// TIA Portal V20 program export: 3 tag tables, 2 data types, 1 data blocks, 4 code blocks (in call order from the OBs), 4 instance data blocks

VAR_GLOBAL   // PLC tag table "IO_Device_PCL_Centralilze_PLC_Functinal_Test_1"
   In_Test_Parameters AT %I100.0 : "IO_Device_Test_Parameters";
   Out_Functinal_Test AT %Q100.0 : "IO_Device_Functinal_Test";
   Voltage_Read_UInt AT %QW160 : UInt;
END_VAR

VAR_GLOBAL   // PLC tag table "IO_PLC_Functinal_Test_1_PLC_Functinal_Test_3"
   In_Functional_Test AT %I300.0 : "IO_Device_Functinal_Test";
   Out_Test_Parameters AT %Q300.0 : "IO_Device_Test_Parameters";
END_VAR

VAR_GLOBAL   // PLC tag table "PLC_Functional_Test"
   Button_Start_Approve AT %I0.0 : Bool;
   Digital_Input_1 AT %I0.1 : Bool;
   Digital_Input_2 AT %I0.2 : Bool;
   Digital_Input_3 AT %I0.3 : Bool;
   Digital_Input_4 AT %I0.4 : Bool;
   Digital_Input_5 AT %I0.5 : Bool;
   Current_Transducer AT %IW64 : Int;
   Voltage_Transducer AT %IW66 : Int;
   Button_Light AT %Q0.0 : Bool;
   Light_Fail_Test AT %Q0.1 : Bool;
   Light_Approve_Test AT %Q0.2 : Bool;
   Digital_Output_3 AT %Q0.3 : Bool;
   Clock_Byte AT %MB0 : Byte;
   Clock_10Hz AT %M0.0 : Bool;
   Clock_5Hz AT %M0.1 : Bool;
   "Clock_2.5Hz" AT %M0.2 : Bool;
   Clock_2Hz AT %M0.3 : Bool;
   "Clock_1.25Hz" AT %M0.4 : Bool;
   Clock_1Hz AT %M0.5 : Bool;
   "Clock_0.625Hz" AT %M0.6 : Bool;
   "Clock_0.5Hz" AT %M0.7 : Bool;
   System_Byte AT %MB1 : Byte;
   FirstScan AT %M1.0 : Bool;
   DiagStatusUpdate AT %M1.1 : Bool;
   AlwaysTRUE AT %M1.2 : Bool;
   AlwaysFALSE AT %M1.3 : Bool;
END_VAR

TYPE "IO_Device_Functinal_Test"
   STRUCT
      Life_Trigger_PLC_Functional_Test_1 : Bool;
      Star_Test_PLC_Functional_Test_1 : Bool;
      Button_PLC_Functional_Test_1 : Bool;
      Electrical_Current_Test_Approved_PLC_Functional_Test_1 : Bool;
      Visual_Test_Approved_PLC_Functional_Test_1 : Bool;
      Electrical_Current_Read_PLC_Functional_Test_1 : UInt;
      Life_Trigger_PLC_Functional_Test_3 : Bool;
      Star_Test_PLC_Functional_Test_3 : Bool;
      Button_PLC_Functional_Test_3 : Bool;
      Electrical_Current_Test_Approved_PLC_Functional_Test_3 : Bool;
      Visual_Test_Approved_PLC_Functional_Test_3 : Bool;
      Electrical_Current_Read_PLC_Functional_Test_3 : UInt;
      Life_Trigger_PLC_Functional_Test_5 : Bool;
      Star_Test_PLC_Functional_Test_5 : Bool;
      Button_PLC_Functional_Test_5 : Bool;
      Electrical_Current_Test_Approved_PLC_Functional_Test_5 : Bool;
      Visual_Test_Approved_PLC_Functional_Test_5 : Bool;
      Electrical_Current_Read_PLC_Functional_Test_5 : UInt;
      Life_Trigger_PLC_Functional_Test_7 : Bool;
      Star_Test_PLC_Functional_Test_7 : Bool;
      Button_PLC_Functional_Test_7 : Bool;
      Electrical_Current_Test_Approved_PLC_Functional_Test_7 : Bool;
      Visual_Test_Approved_PLC_Functional_Test_7 : Bool;
      Electrical_Current_Read_PLC_Functional_Test_7 : UInt;
      Life_Trigger_PLC_Functional_Test_9 : Bool;
      Star_Test_PLC_Functional_Test_9 : Bool;
      Button_PLC_Functional_Test_9 : Bool;
      Electrical_Current_Test_Approved_PLC_Functional_Test_9 : Bool;
      Visual_Test_Approved_PLC_Functional_Test_9 : Bool;
      Electrical_Current_Read_PLC_Functional_Test_9 : UInt;
      Life_Trigger_PLC_Functional_Test_11 : Bool;
      Star_Test_PLC_Functional_Test_11 : Bool;
      Button_PLC_Functional_Test_11 : Bool;
      Electrical_Current_Test_Approved_PLC_Functional_Test_11 : Bool;
      Visual_Test_Approved_PLC_Functional_Test_11 : Bool;
      Electrical_Current_Read_PLC_Functional_Test_11 : UInt;
      Life_Trigger_PLC_Functional_Test_13 : Bool;
      Star_Test_PLC_Functional_Test_13 : Bool;
      Button_PLC_Functional_Test_13 : Bool;
      Electrical_Current_Test_Approved_PLC_Functional_Test_13 : Bool;
      Visual_Test_Approved_PLC_Functional_Test_13 : Bool;
      Electrical_Current_Read_PLC_Functional_Test_13 : UInt;
      Life_Trigger_PLC_Functional_Test_15 : Bool;
      Star_Test_PLC_Functional_Test_15 : Bool;
      Button_PLC_Functional_Test_15 : Bool;
      Electrical_Current_Test_Approved_PLC_Functional_Test_15 : Bool;
      Visual_Test_Approved_PLC_Functional_Test_15 : Bool;
      Electrical_Current_Read_PLC_Functional_Test_15 : UInt;
      Life_Trigger_PLC_Functional_Test_17 : Bool;
      Star_Test_PLC_Functional_Test_17 : Bool;
      Button_PLC_Functional_Test_17 : Bool;
      Electrical_Current_Test_Approved_PLC_Functional_Test_17 : Bool;
      Visual_Test_Approved_PLC_Functional_Test_17 : Bool;
      Electrical_Current_Read_PLC_Functional_Test_17 : UInt;
      Life_Trigger_PLC_Functional_Test_19 : Bool;
      Star_Test_PLC_Functional_Test_19 : Bool;
      Button_PLC_Functional_Test_19 : Bool;
      Electrical_Current_Test_Approved_PLC_Functional_Test_19 : Bool;
      Visual_Test_Approved_PLC_Functional_Test_19 : Bool;
      Electrical_Current_Read_PLC_Functional_Test_19 : UInt;
      Life_Trigger_PLC_Functional_Test_21 : Bool;
      Star_Test_PLC_Functional_Test_21 : Bool;
      Button_PLC_Functional_Test_21 : Bool;
      Electrical_Current_Test_Approved_PLC_Functional_Test_21 : Bool;
      Visual_Test_Approved_PLC_Functional_Test_21 : Bool;
      Electrical_Current_Read_PLC_Functional_Test_21 : UInt;
      Life_Trigger_PLC_Functional_Test_23 : Bool;
      Star_Test_PLC_Functional_Test_23 : Bool;
      Button_PLC_Functional_Test_23 : Bool;
      Electrical_Current_Test_Approved_PLC_Functional_Test_23 : Bool;
      Visual_Test_Approved_PLC_Functional_Test_23 : Bool;
      Electrical_Current_Read_PLC_Functional_Test_23 : UInt;
      Life_Trigger_PLC_Functional_Test_25 : Bool;
      Star_Test_PLC_Functional_Test_25 : Bool;
      Button_PLC_Functional_Test_25 : Bool;
      Electrical_Current_Test_Approved_PLC_Functional_Test_25 : Bool;
      Visual_Test_Approved_PLC_Functional_Test_25 : Bool;
      Electrical_Current_Read_PLC_Functional_Test_25 : UInt;
      Life_Trigger_PLC_Functional_Test_27 : Bool;
      Star_Test_PLC_Functional_Test_27 : Bool;
      Button_PLC_Functional_Test_27 : Bool;
      Electrical_Current_Test_Approved_PLC_Functional_Test_27 : Bool;
      Visual_Test_Approved_PLC_Functional_Test_27 : Bool;
      Electrical_Current_Read_PLC_Functional_Test_27 : UInt;
      Life_Trigger_PLC_Functional_Test_29 : Bool;
      Star_Test_PLC_Functional_Test_29 : Bool;
      Button_PLC_Functional_Test_29 : Bool;
      Electrical_Current_Test_Approved_PLC_Functional_Test_29 : Bool;
      Visual_Test_Approved_PLC_Functional_Test_29 : Bool;
      Electrical_Current_Read_PLC_Functional_Test_29 : UInt;
   END_STRUCT;
END_TYPE

TYPE "IO_Device_Test_Parameters"
   STRUCT
      Reset_PLC_Functional_Test_1 : Bool;
      Reset_PLC_Functional_Test_3 : Bool;
      Reset_PLC_Functional_Test_5 : Bool;
      Reset_PLC_Functional_Test_7 : Bool;
      Reset_PLC_Functional_Test_9 : Bool;
      Reset_PLC_Functional_Test_11 : Bool;
      Reset_PLC_Functional_Test_13 : Bool;
      Reset_PLC_Functional_Test_15 : Bool;
      Reset_PLC_Functional_Test_17 : Bool;
      Reset_PLC_Functional_Test_19 : Bool;
      Reset_PLC_Functional_Test_21 : Bool;
      Reset_PLC_Functional_Test_23 : Bool;
      Reset_PLC_Functional_Test_25 : Bool;
      Reset_PLC_Functional_Test_27 : Bool;
      Reset_PLC_Functional_Test_29 : Bool;
      Status : Bool;
      Voltage_Read : UInt;
      Min_Electrical_Current : UInt;
      Max_Electrical_Current : UInt;
      Time_End_Electrical_Current_Test : Time;
      Time_Start_Visual_Test : Time;
   END_STRUCT;
END_TYPE

DATA_BLOCK "DB_Test_Water_Foutain"   // DB4
{ S7_Optimized_Access := 'TRUE' }
// stored: MemoryReserve 100
   VAR
      Star_Functional_Test : Bool;
      Reset_Functional_Test : Bool;
      Electrical_Current_Test_Approved : Bool;
      Visual_Test_Approved_PLC : Bool;
   END_VAR
BEGIN
END_DATA_BLOCK

ORGANIZATION_BLOCK "Main"   // OB1, LAD, ProgramCycle
TITLE = "Main Program Sweep (Cycle)"
{ S7_Optimized_Access := 'TRUE' }
// stored: SetENOAutomatically false
   VAR_INPUT
      Initial_Call : Bool;   // Initial call of this OB
      Remanence : Bool;   // =True, if remanent data are available
   END_VAR
   VAR CONSTANT
      Test_Station : SInt := 1;
      Total_Number_Test_Stations : SInt := 25;
   END_VAR
BEGIN

REGION Network 1: Digital Inputs
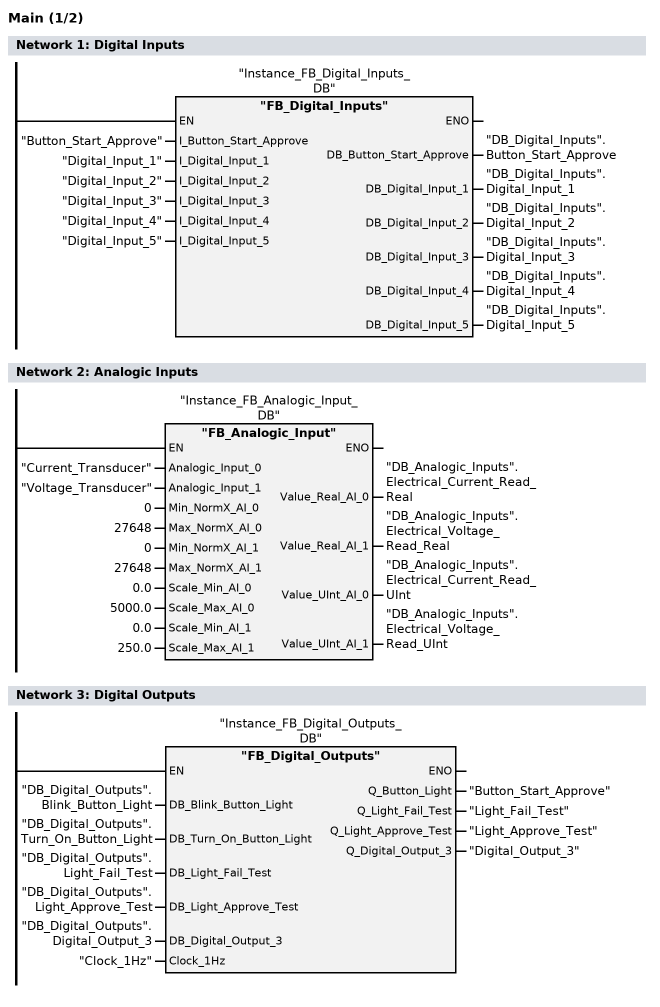
   RUNG wire#powerrail
      "Instance_FB_Digital_Inputs_DB"(I_Button_Start_Approve := "Button_Start_Approve", I_Digital_Input_1 := "Digital_Input_1", I_Digital_Input_2 := "Digital_Input_2", I_Digital_Input_3 := "Digital_Input_3", I_Digital_Input_4 := "Digital_Input_4", I_Digital_Input_5 := "Digital_Input_5", DB_Button_Start_Approve => "DB_Digital_Inputs".Button_Start_Approve, DB_Digital_Input_1 => "DB_Digital_Inputs".Digital_Input_1, DB_Digital_Input_2 => "DB_Digital_Inputs".Digital_Input_2, DB_Digital_Input_3 => "DB_Digital_Inputs".Digital_Input_3, DB_Digital_Input_4 => "DB_Digital_Inputs".Digital_Input_4, DB_Digital_Input_5 => "DB_Digital_Inputs".Digital_Input_5)
   END_RUNG
   // the same network as SCL:
   "Instance_FB_Digital_Inputs_DB"(I_Button_Start_Approve := "Button_Start_Approve",   // "FB_Digital_Inputs"
                           I_Digital_Input_1 := "Digital_Input_1",
                           I_Digital_Input_2 := "Digital_Input_2",
                           I_Digital_Input_3 := "Digital_Input_3",
                           I_Digital_Input_4 := "Digital_Input_4",
                           I_Digital_Input_5 := "Digital_Input_5",
                           DB_Button_Start_Approve => "DB_Digital_Inputs".Button_Start_Approve,
                           DB_Digital_Input_1 => "DB_Digital_Inputs".Digital_Input_1,
                           DB_Digital_Input_2 => "DB_Digital_Inputs".Digital_Input_2,
                           DB_Digital_Input_3 => "DB_Digital_Inputs".Digital_Input_3,
                           DB_Digital_Input_4 => "DB_Digital_Inputs".Digital_Input_4,
                           DB_Digital_Input_5 => "DB_Digital_Inputs".Digital_Input_5);
END_REGION

REGION Network 2: Analogic Inputs
   RUNG wire#powerrail
      "Instance_FB_Analogic_Input_DB"(Analogic_Input_0 := "Current_Transducer", Analogic_Input_1 := "Voltage_Transducer", Min_NormX_AI_0 := 0, Max_NormX_AI_0 := 27648, Min_NormX_AI_1 := 0, Max_NormX_AI_1 := 27648, Scale_Min_AI_0 := 0.0, Scale_Max_AI_0 := 5000.0, Scale_Min_AI_1 := 0.0, Scale_Max_AI_1 := 250.0, Value_Real_AI_0 => "DB_Analogic_Inputs".Electrical_Current_Read_Real, Value_Real_AI_1 => "DB_Analogic_Inputs".Electrical_Voltage_Read_Real, Value_UInt_AI_0 => "DB_Analogic_Inputs".Electrical_Current_Read_UInt, Value_UInt_AI_1 => "DB_Analogic_Inputs".Electrical_Voltage_Read_UInt)
   END_RUNG
   // the same network as SCL:
   "Instance_FB_Analogic_Input_DB"(Analogic_Input_0 := "Current_Transducer",   // "FB_Analogic_Input"
                           Analogic_Input_1 := "Voltage_Transducer",
                           Min_NormX_AI_0 := 0,
                           Max_NormX_AI_0 := 27648,
                           Min_NormX_AI_1 := 0,
                           Max_NormX_AI_1 := 27648,
                           Scale_Min_AI_0 := 0.0,
                           Scale_Max_AI_0 := 5000.0,
                           Scale_Min_AI_1 := 0.0,
                           Scale_Max_AI_1 := 250.0,
                           Value_Real_AI_0 => "DB_Analogic_Inputs".Electrical_Current_Read_Real,
                           Value_Real_AI_1 => "DB_Analogic_Inputs".Electrical_Voltage_Read_Real,
                           Value_UInt_AI_0 => "DB_Analogic_Inputs".Electrical_Current_Read_UInt,
                           Value_UInt_AI_1 => "DB_Analogic_Inputs".Electrical_Voltage_Read_UInt);
END_REGION

REGION Network 3: Digital Outputs
   RUNG wire#powerrail
      "Instance_FB_Digital_Outputs_DB"(DB_Blink_Button_Light := "DB_Digital_Outputs".Blink_Button_Light, DB_Turn_On_Button_Light := "DB_Digital_Outputs".Turn_On_Button_Light, DB_Light_Fail_Test := "DB_Digital_Outputs".Light_Fail_Test, DB_Light_Approve_Test := "DB_Digital_Outputs".Light_Approve_Test, DB_Digital_Output_3 := "DB_Digital_Outputs".Digital_Output_3, Clock_1Hz := "Clock_1Hz", Q_Button_Light => "Button_Start_Approve", Q_Light_Fail_Test => "Light_Fail_Test", Q_Light_Approve_Test => "Light_Approve_Test", Q_Digital_Output_3 => "Digital_Output_3")
   END_RUNG
   // the same network as SCL:
   "Instance_FB_Digital_Outputs_DB"(DB_Blink_Button_Light := "DB_Digital_Outputs".Blink_Button_Light,   // "FB_Digital_Outputs"
                           DB_Turn_On_Button_Light := "DB_Digital_Outputs".Turn_On_Button_Light,
                           DB_Light_Fail_Test := "DB_Digital_Outputs".Light_Fail_Test,
                           DB_Light_Approve_Test := "DB_Digital_Outputs".Light_Approve_Test,
                           DB_Digital_Output_3 := "DB_Digital_Outputs".Digital_Output_3,
                           Clock_1Hz := "Clock_1Hz",
                           Q_Button_Light => "Button_Start_Approve",
                           Q_Light_Fail_Test => "Light_Fail_Test",
                           Q_Light_Approve_Test => "Light_Approve_Test",
                           Q_Digital_Output_3 => "Digital_Output_3");
END_REGION

REGION Network 4: IO Device
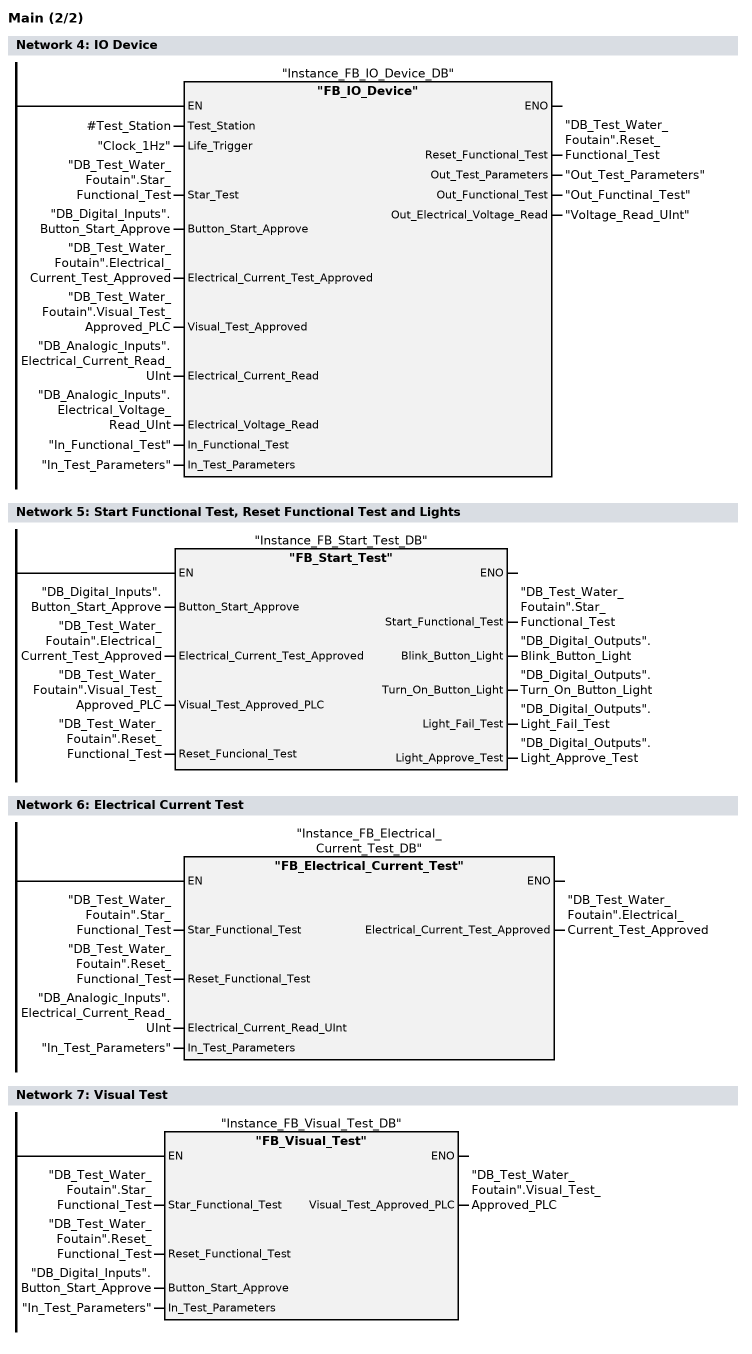
   RUNG wire#powerrail
      "Instance_FB_IO_Device_DB"(Test_Station := #Test_Station, Life_Trigger := "Clock_1Hz", Star_Test := "DB_Test_Water_Foutain".Star_Functional_Test, Button_Start_Approve := "DB_Digital_Inputs".Button_Start_Approve, Electrical_Current_Test_Approved := "DB_Test_Water_Foutain".Electrical_Current_Test_Approved, Visual_Test_Approved := "DB_Test_Water_Foutain".Visual_Test_Approved_PLC, Electrical_Current_Read := "DB_Analogic_Inputs".Electrical_Current_Read_UInt, Electrical_Voltage_Read := "DB_Analogic_Inputs".Electrical_Voltage_Read_UInt, In_Functional_Test := "In_Functional_Test", In_Test_Parameters := "In_Test_Parameters", Reset_Functional_Test => "DB_Test_Water_Foutain".Reset_Functional_Test, Out_Test_Parameters => "Out_Test_Parameters", Out_Functional_Test => "Out_Functinal_Test", Out_Electrical_Voltage_Read => "Voltage_Read_UInt")
   END_RUNG
   // the same network as SCL:
   "Instance_FB_IO_Device_DB"(Test_Station := #Test_Station,   // "FB_IO_Device"
                           Life_Trigger := "Clock_1Hz",
                           Star_Test := "DB_Test_Water_Foutain".Star_Functional_Test,
                           Button_Start_Approve := "DB_Digital_Inputs".Button_Start_Approve,
                           Electrical_Current_Test_Approved := "DB_Test_Water_Foutain".Electrical_Current_Test_Approved,
                           Visual_Test_Approved := "DB_Test_Water_Foutain".Visual_Test_Approved_PLC,
                           Electrical_Current_Read := "DB_Analogic_Inputs".Electrical_Current_Read_UInt,
                           Electrical_Voltage_Read := "DB_Analogic_Inputs".Electrical_Voltage_Read_UInt,
                           In_Functional_Test := "In_Functional_Test",
                           In_Test_Parameters := "In_Test_Parameters",
                           Reset_Functional_Test => "DB_Test_Water_Foutain".Reset_Functional_Test,
                           Out_Test_Parameters => "Out_Test_Parameters",
                           Out_Functional_Test => "Out_Functinal_Test",
                           Out_Electrical_Voltage_Read => "Voltage_Read_UInt");
END_REGION

REGION Network 5: Start Functional Test, Reset Functional Test and Lights
   RUNG wire#powerrail
      "Instance_FB_Start_Test_DB"(Button_Start_Approve := "DB_Digital_Inputs".Button_Start_Approve, Electrical_Current_Test_Approved := "DB_Test_Water_Foutain".Electrical_Current_Test_Approved, Visual_Test_Approved_PLC := "DB_Test_Water_Foutain".Visual_Test_Approved_PLC, Reset_Funcional_Test := "DB_Test_Water_Foutain".Reset_Functional_Test, Start_Functional_Test => "DB_Test_Water_Foutain".Star_Functional_Test, Blink_Button_Light => "DB_Digital_Outputs".Blink_Button_Light, Turn_On_Button_Light => "DB_Digital_Outputs".Turn_On_Button_Light, Light_Fail_Test => "DB_Digital_Outputs".Light_Fail_Test, Light_Approve_Test => "DB_Digital_Outputs".Light_Approve_Test)
   END_RUNG
   // the same network as SCL:
   "Instance_FB_Start_Test_DB"(Button_Start_Approve := "DB_Digital_Inputs".Button_Start_Approve,   // "FB_Start_Test"
                           Electrical_Current_Test_Approved := "DB_Test_Water_Foutain".Electrical_Current_Test_Approved,
                           Visual_Test_Approved_PLC := "DB_Test_Water_Foutain".Visual_Test_Approved_PLC,
                           Reset_Funcional_Test := "DB_Test_Water_Foutain".Reset_Functional_Test,
                           Start_Functional_Test => "DB_Test_Water_Foutain".Star_Functional_Test,
                           Blink_Button_Light => "DB_Digital_Outputs".Blink_Button_Light,
                           Turn_On_Button_Light => "DB_Digital_Outputs".Turn_On_Button_Light,
                           Light_Fail_Test => "DB_Digital_Outputs".Light_Fail_Test,
                           Light_Approve_Test => "DB_Digital_Outputs".Light_Approve_Test);
END_REGION

REGION Network 6: Electrical Current Test
   RUNG wire#powerrail
      "Instance_FB_Electrical_Current_Test_DB"(Star_Functional_Test := "DB_Test_Water_Foutain".Star_Functional_Test, Reset_Functional_Test := "DB_Test_Water_Foutain".Reset_Functional_Test, Electrical_Current_Read_UInt := "DB_Analogic_Inputs".Electrical_Current_Read_UInt, In_Test_Parameters := "In_Test_Parameters", Electrical_Current_Test_Approved => "DB_Test_Water_Foutain".Electrical_Current_Test_Approved)
   END_RUNG
   // the same network as SCL:
   "Instance_FB_Electrical_Current_Test_DB"(Star_Functional_Test := "DB_Test_Water_Foutain".Star_Functional_Test,   // "FB_Electrical_Current_Test"
                           Reset_Functional_Test := "DB_Test_Water_Foutain".Reset_Functional_Test,
                           Electrical_Current_Read_UInt := "DB_Analogic_Inputs".Electrical_Current_Read_UInt,
                           In_Test_Parameters := "In_Test_Parameters",
                           Electrical_Current_Test_Approved => "DB_Test_Water_Foutain".Electrical_Current_Test_Approved);
END_REGION

REGION Network 7: Visual Test
   RUNG wire#powerrail
      "Instance_FB_Visual_Test_DB"(Star_Functional_Test := "DB_Test_Water_Foutain".Star_Functional_Test, Reset_Functional_Test := "DB_Test_Water_Foutain".Reset_Functional_Test, Button_Start_Approve := "DB_Digital_Inputs".Button_Start_Approve, In_Test_Parameters := "In_Test_Parameters", Visual_Test_Approved_PLC => "DB_Test_Water_Foutain".Visual_Test_Approved_PLC)
   END_RUNG
   // the same network as SCL:
   "Instance_FB_Visual_Test_DB"(Star_Functional_Test := "DB_Test_Water_Foutain".Star_Functional_Test,   // "FB_Visual_Test"
                           Reset_Functional_Test := "DB_Test_Water_Foutain".Reset_Functional_Test,
                           Button_Start_Approve := "DB_Digital_Inputs".Button_Start_Approve,
                           In_Test_Parameters := "In_Test_Parameters",
                           Visual_Test_Approved_PLC => "DB_Test_Water_Foutain".Visual_Test_Approved_PLC);
END_REGION
END_ORGANIZATION_BLOCK

FUNCTION_BLOCK "FB_IO_Device"   // FB4, LAD
{ S7_Optimized_Access := 'TRUE' }
// stored: MemoryReserve 100, SetENOAutomatically false
   VAR_INPUT
      Test_Station : SInt;
      Life_Trigger : Bool;
      Star_Test : Bool;
      Button_Start_Approve : Bool;
      Electrical_Current_Test_Approved : Bool;
      Visual_Test_Approved : Bool;
      Electrical_Current_Read : UInt;
      Electrical_Voltage_Read : UInt;
      In_Functional_Test : "IO_Device_Functinal_Test";
      In_Test_Parameters : "IO_Device_Test_Parameters";
   END_VAR
   VAR_OUTPUT
      Reset_Functional_Test : Bool;
      Out_Test_Parameters : "IO_Device_Test_Parameters";
      Out_Functional_Test : "IO_Device_Functinal_Test";
      Out_Electrical_Voltage_Read : UInt;
   END_VAR
   VAR_TEMP   // added for the SCL form of the ladder/FBD networks
      _w1 : Bool;
   END_VAR
BEGIN

REGION Network 1: Test Parameters
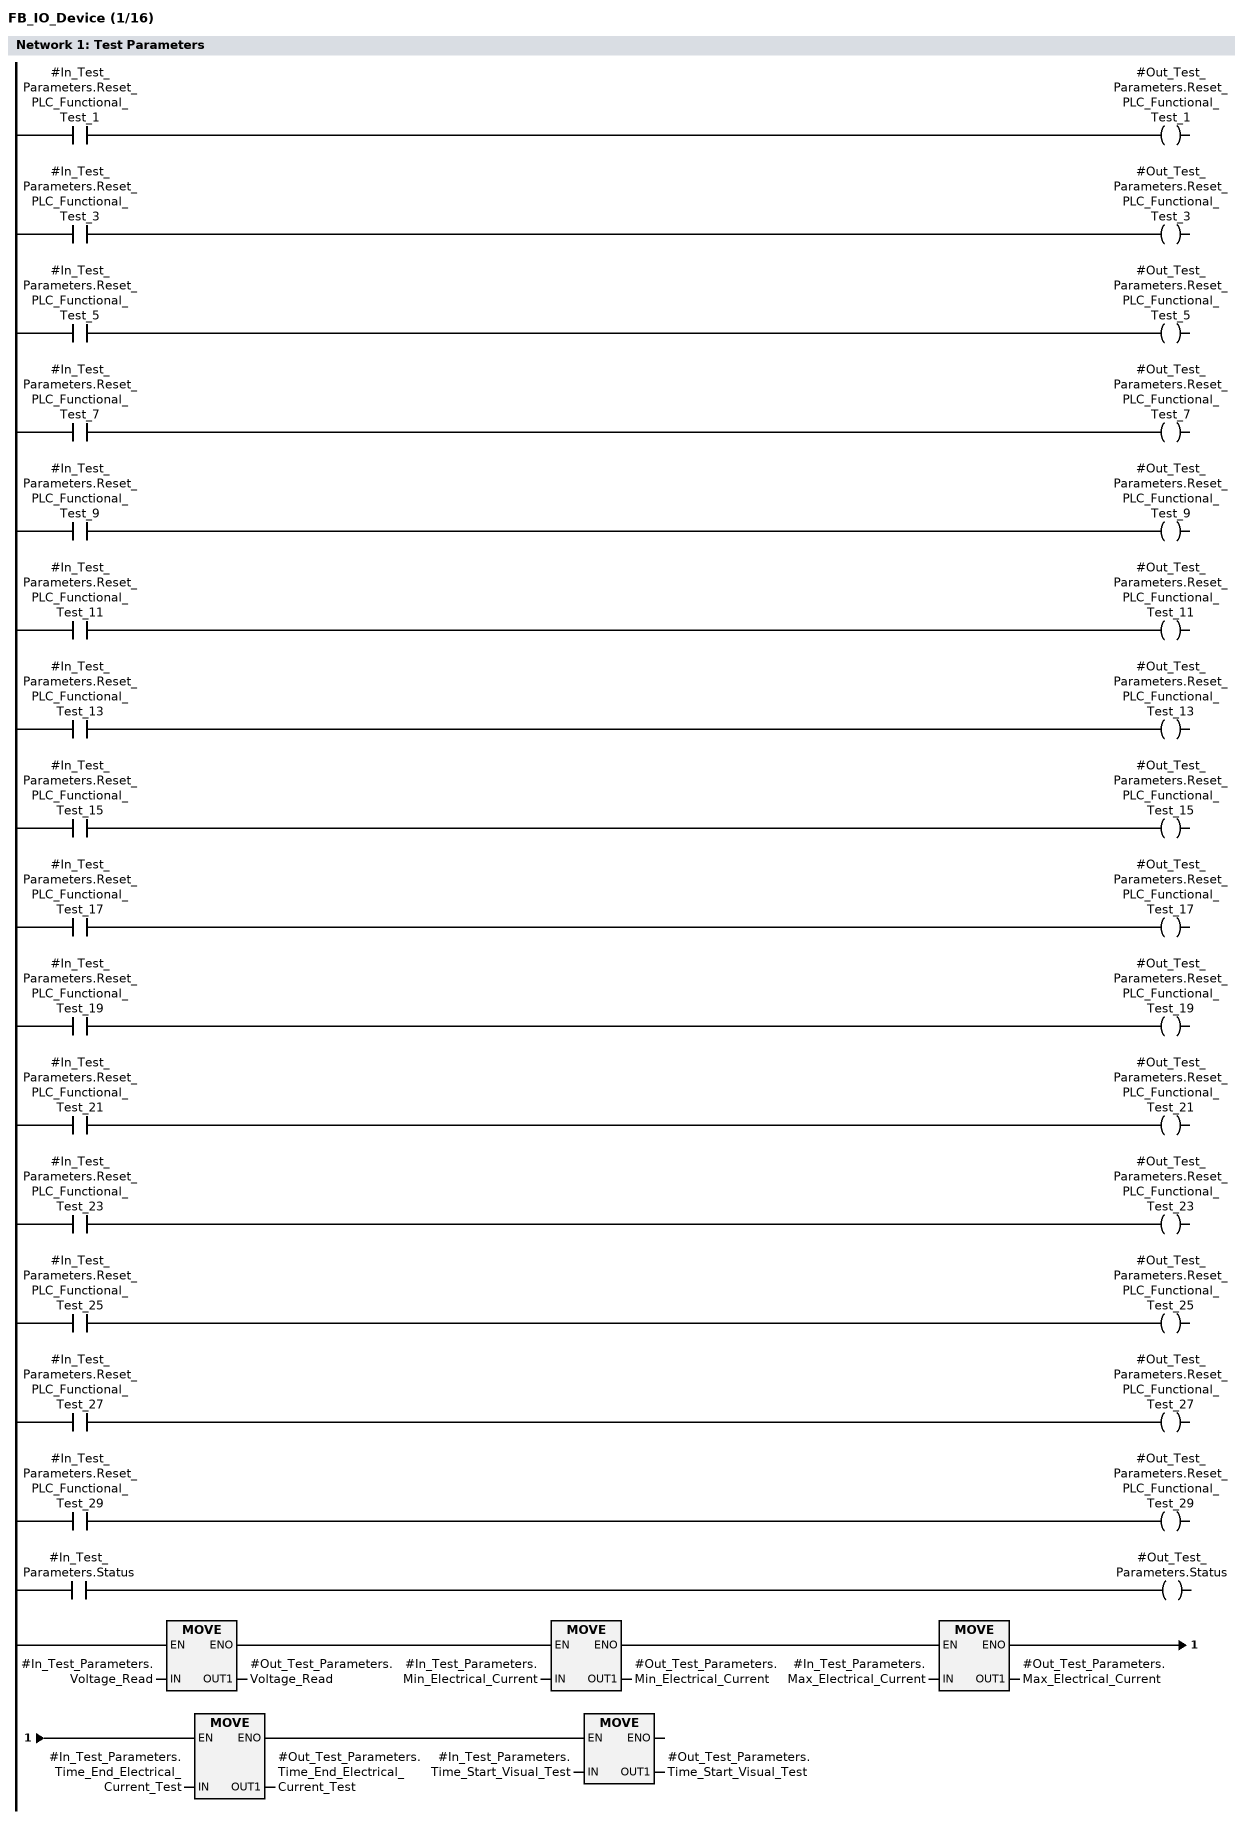
   RUNG wire#powerrail
      Contact( #In_Test_Parameters.Reset_PLC_Functional_Test_1 )
      Coil( #Out_Test_Parameters.Reset_PLC_Functional_Test_1 )
   END_RUNG
   RUNG wire#powerrail
      Contact( #In_Test_Parameters.Reset_PLC_Functional_Test_3 )
      Coil( #Out_Test_Parameters.Reset_PLC_Functional_Test_3 )
   END_RUNG
   RUNG wire#powerrail
      Contact( #In_Test_Parameters.Reset_PLC_Functional_Test_5 )
      Coil( #Out_Test_Parameters.Reset_PLC_Functional_Test_5 )
   END_RUNG
   RUNG wire#powerrail
      Contact( #In_Test_Parameters.Reset_PLC_Functional_Test_7 )
      Coil( #Out_Test_Parameters.Reset_PLC_Functional_Test_7 )
   END_RUNG
   RUNG wire#powerrail
      Contact( #In_Test_Parameters.Reset_PLC_Functional_Test_9 )
      Coil( #Out_Test_Parameters.Reset_PLC_Functional_Test_9 )
   END_RUNG
   RUNG wire#powerrail
      Contact( #In_Test_Parameters.Reset_PLC_Functional_Test_11 )
      Coil( #Out_Test_Parameters.Reset_PLC_Functional_Test_11 )
   END_RUNG
   RUNG wire#powerrail
      Contact( #In_Test_Parameters.Reset_PLC_Functional_Test_13 )
      Coil( #Out_Test_Parameters.Reset_PLC_Functional_Test_13 )
   END_RUNG
   RUNG wire#powerrail
      Contact( #In_Test_Parameters.Reset_PLC_Functional_Test_15 )
      Coil( #Out_Test_Parameters.Reset_PLC_Functional_Test_15 )
   END_RUNG
   RUNG wire#powerrail
      Contact( #In_Test_Parameters.Reset_PLC_Functional_Test_17 )
      Coil( #Out_Test_Parameters.Reset_PLC_Functional_Test_17 )
   END_RUNG
   RUNG wire#powerrail
      Contact( #In_Test_Parameters.Reset_PLC_Functional_Test_19 )
      Coil( #Out_Test_Parameters.Reset_PLC_Functional_Test_19 )
   END_RUNG
   RUNG wire#powerrail
      Contact( #In_Test_Parameters.Reset_PLC_Functional_Test_21 )
      Coil( #Out_Test_Parameters.Reset_PLC_Functional_Test_21 )
   END_RUNG
   RUNG wire#powerrail
      Contact( #In_Test_Parameters.Reset_PLC_Functional_Test_23 )
      Coil( #Out_Test_Parameters.Reset_PLC_Functional_Test_23 )
   END_RUNG
   RUNG wire#powerrail
      Contact( #In_Test_Parameters.Reset_PLC_Functional_Test_25 )
      Coil( #Out_Test_Parameters.Reset_PLC_Functional_Test_25 )
   END_RUNG
   RUNG wire#powerrail
      Contact( #In_Test_Parameters.Reset_PLC_Functional_Test_27 )
      Coil( #Out_Test_Parameters.Reset_PLC_Functional_Test_27 )
   END_RUNG
   RUNG wire#powerrail
      Contact( #In_Test_Parameters.Reset_PLC_Functional_Test_29 )
      Coil( #Out_Test_Parameters.Reset_PLC_Functional_Test_29 )
   END_RUNG
   RUNG wire#powerrail
      Contact( #In_Test_Parameters.Status )
      Coil( #Out_Test_Parameters.Status )
   END_RUNG
   RUNG wire#powerrail
      Move(in := #In_Test_Parameters.Voltage_Read, out1 => #Out_Test_Parameters.Voltage_Read)
      Move(in := #In_Test_Parameters.Min_Electrical_Current, out1 => #Out_Test_Parameters.Min_Electrical_Current)
      Move(in := #In_Test_Parameters.Max_Electrical_Current, out1 => #Out_Test_Parameters.Max_Electrical_Current)
      Move(in := #In_Test_Parameters.Time_End_Electrical_Current_Test, out1 => #Out_Test_Parameters.Time_End_Electrical_Current_Test)
      Move(in := #In_Test_Parameters.Time_Start_Visual_Test, out1 => #Out_Test_Parameters.Time_Start_Visual_Test)
   END_RUNG
   // the same network as SCL:
   #Out_Test_Parameters.Reset_PLC_Functional_Test_1 := #In_Test_Parameters.Reset_PLC_Functional_Test_1;
   #Out_Test_Parameters.Reset_PLC_Functional_Test_3 := #In_Test_Parameters.Reset_PLC_Functional_Test_3;
   #Out_Test_Parameters.Reset_PLC_Functional_Test_5 := #In_Test_Parameters.Reset_PLC_Functional_Test_5;
   #Out_Test_Parameters.Reset_PLC_Functional_Test_7 := #In_Test_Parameters.Reset_PLC_Functional_Test_7;
   #Out_Test_Parameters.Reset_PLC_Functional_Test_9 := #In_Test_Parameters.Reset_PLC_Functional_Test_9;
   #Out_Test_Parameters.Reset_PLC_Functional_Test_11 := #In_Test_Parameters.Reset_PLC_Functional_Test_11;
   #Out_Test_Parameters.Reset_PLC_Functional_Test_13 := #In_Test_Parameters.Reset_PLC_Functional_Test_13;
   #Out_Test_Parameters.Reset_PLC_Functional_Test_15 := #In_Test_Parameters.Reset_PLC_Functional_Test_15;
   #Out_Test_Parameters.Reset_PLC_Functional_Test_17 := #In_Test_Parameters.Reset_PLC_Functional_Test_17;
   #Out_Test_Parameters.Reset_PLC_Functional_Test_19 := #In_Test_Parameters.Reset_PLC_Functional_Test_19;
   #Out_Test_Parameters.Reset_PLC_Functional_Test_21 := #In_Test_Parameters.Reset_PLC_Functional_Test_21;
   #Out_Test_Parameters.Reset_PLC_Functional_Test_23 := #In_Test_Parameters.Reset_PLC_Functional_Test_23;
   #Out_Test_Parameters.Reset_PLC_Functional_Test_25 := #In_Test_Parameters.Reset_PLC_Functional_Test_25;
   #Out_Test_Parameters.Reset_PLC_Functional_Test_27 := #In_Test_Parameters.Reset_PLC_Functional_Test_27;
   #Out_Test_Parameters.Reset_PLC_Functional_Test_29 := #In_Test_Parameters.Reset_PLC_Functional_Test_29;
   #Out_Test_Parameters.Status := #In_Test_Parameters.Status;
   #Out_Test_Parameters.Voltage_Read := #In_Test_Parameters.Voltage_Read;
   #Out_Test_Parameters.Min_Electrical_Current := #In_Test_Parameters.Min_Electrical_Current;
   #Out_Test_Parameters.Max_Electrical_Current := #In_Test_Parameters.Max_Electrical_Current;
   #Out_Test_Parameters.Time_End_Electrical_Current_Test := #In_Test_Parameters.Time_End_Electrical_Current_Test;
   #Out_Test_Parameters.Time_Start_Visual_Test := #In_Test_Parameters.Time_Start_Visual_Test;
END_REGION

REGION Network 2: Functional Test Station 1
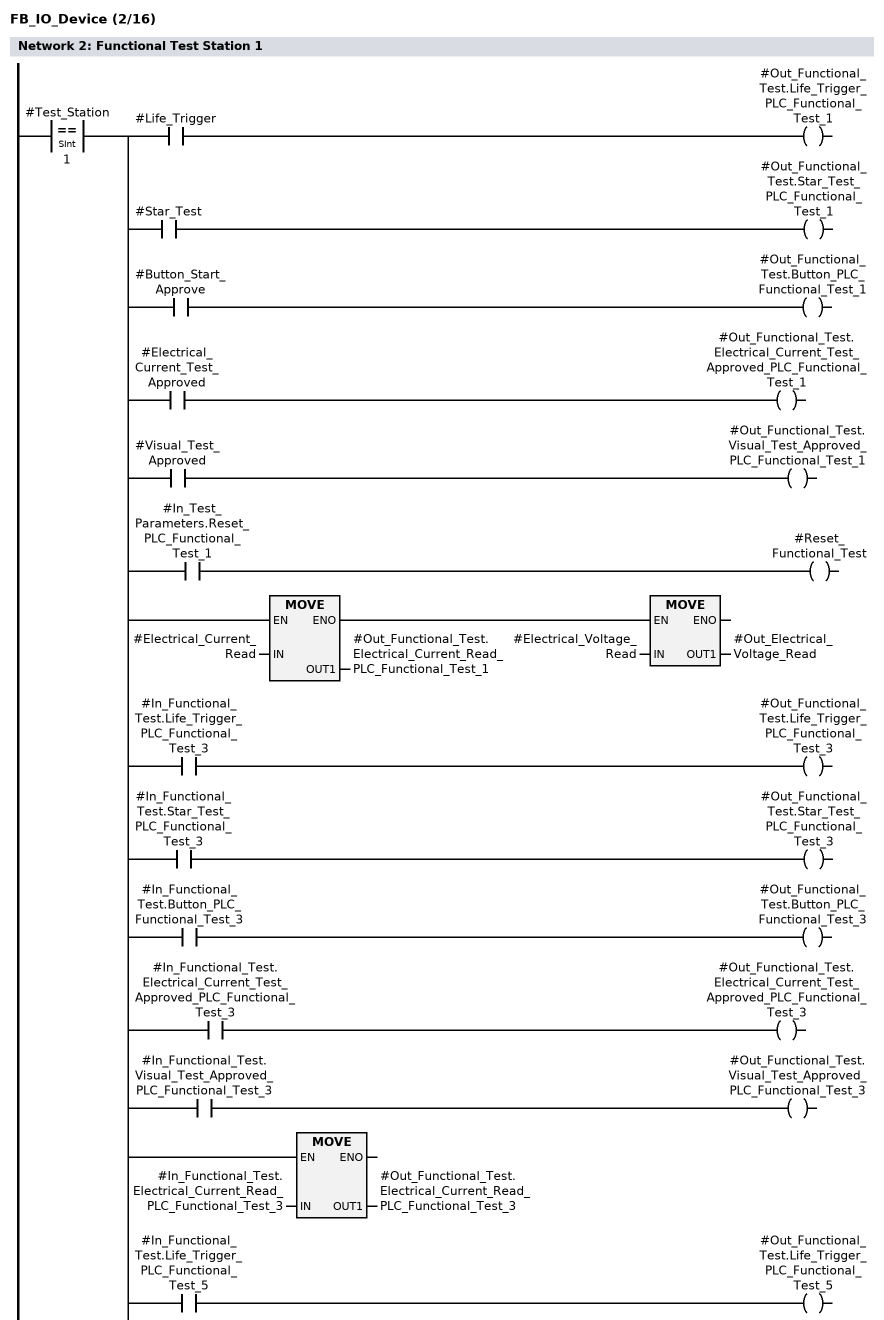
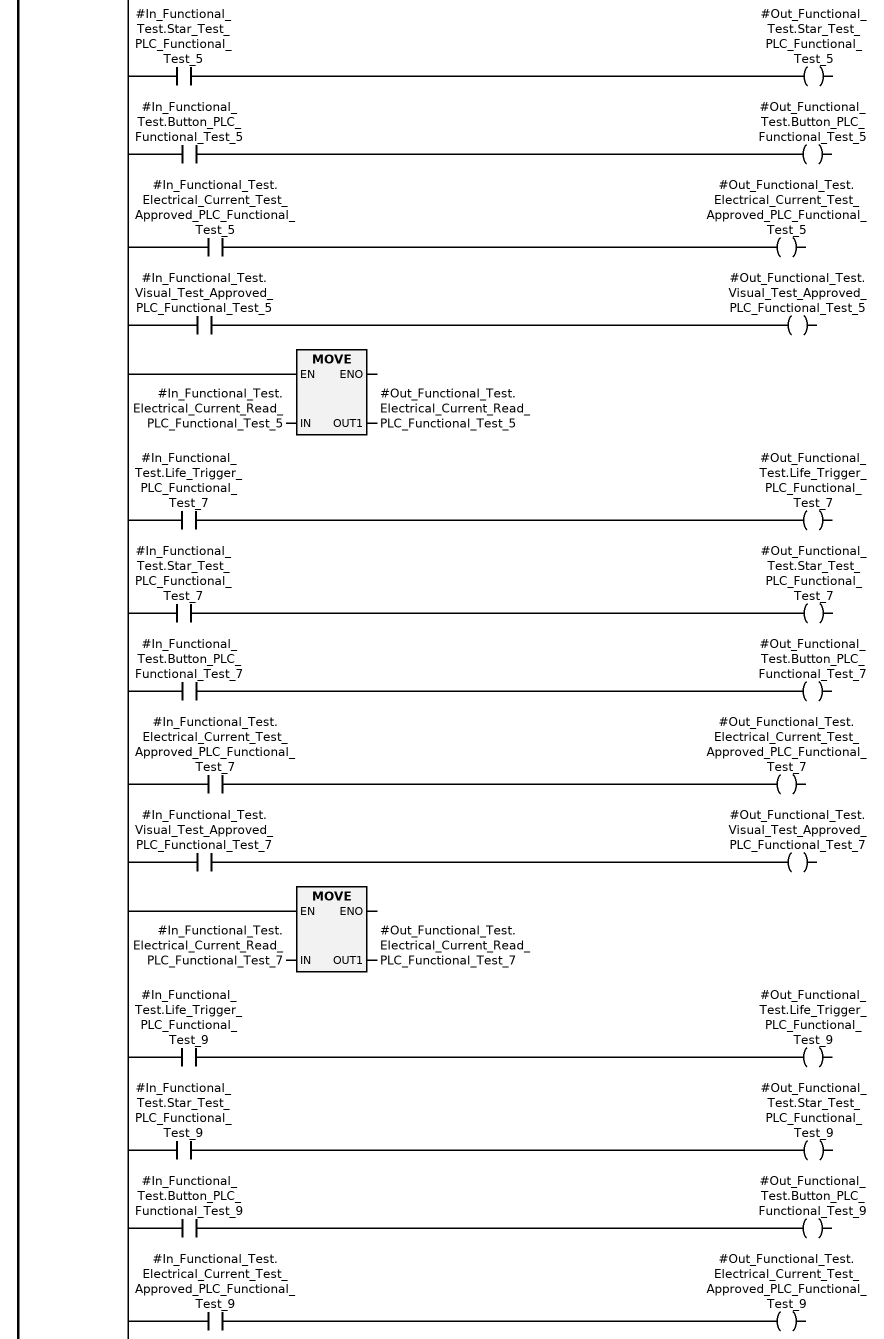
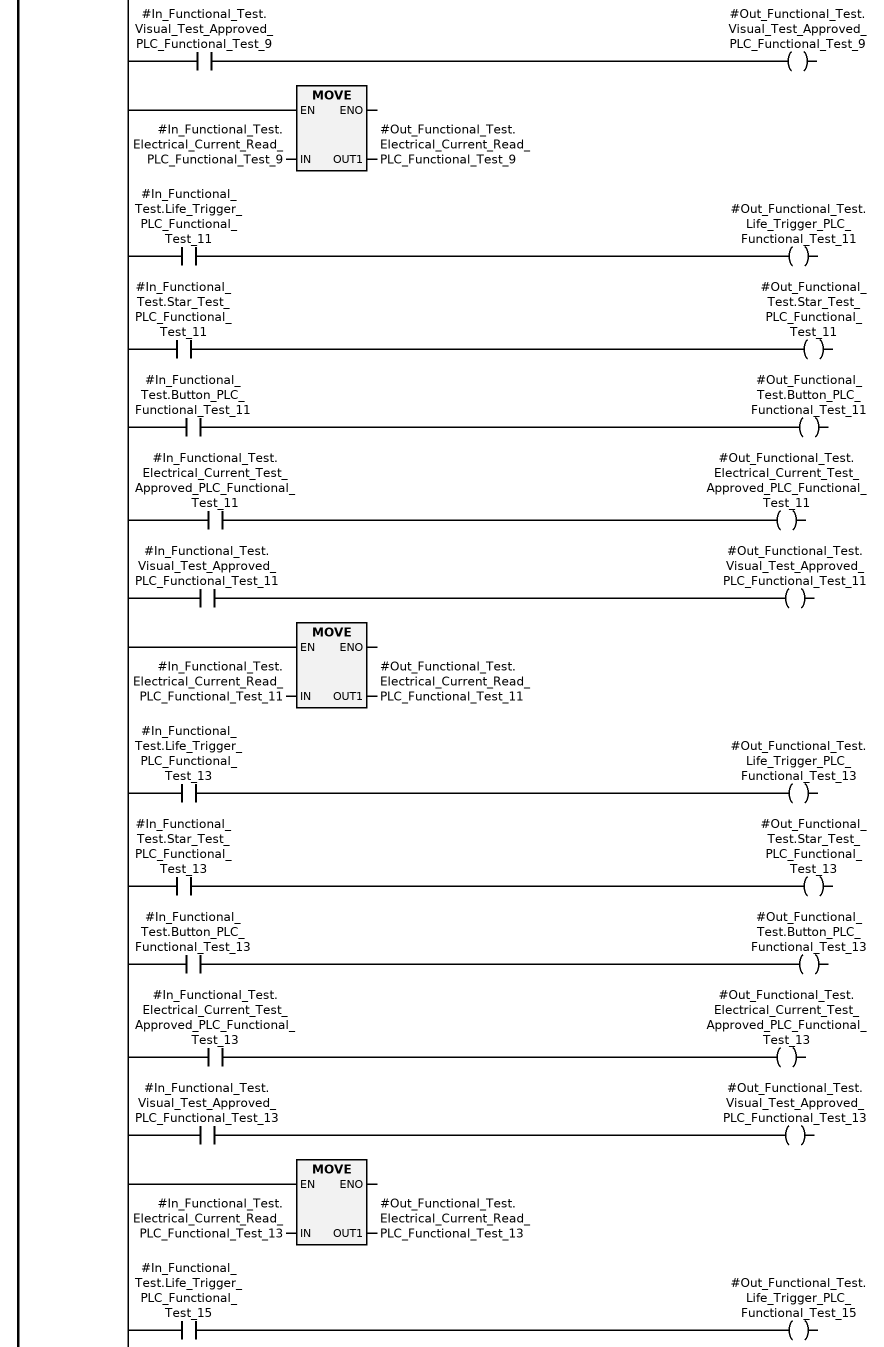
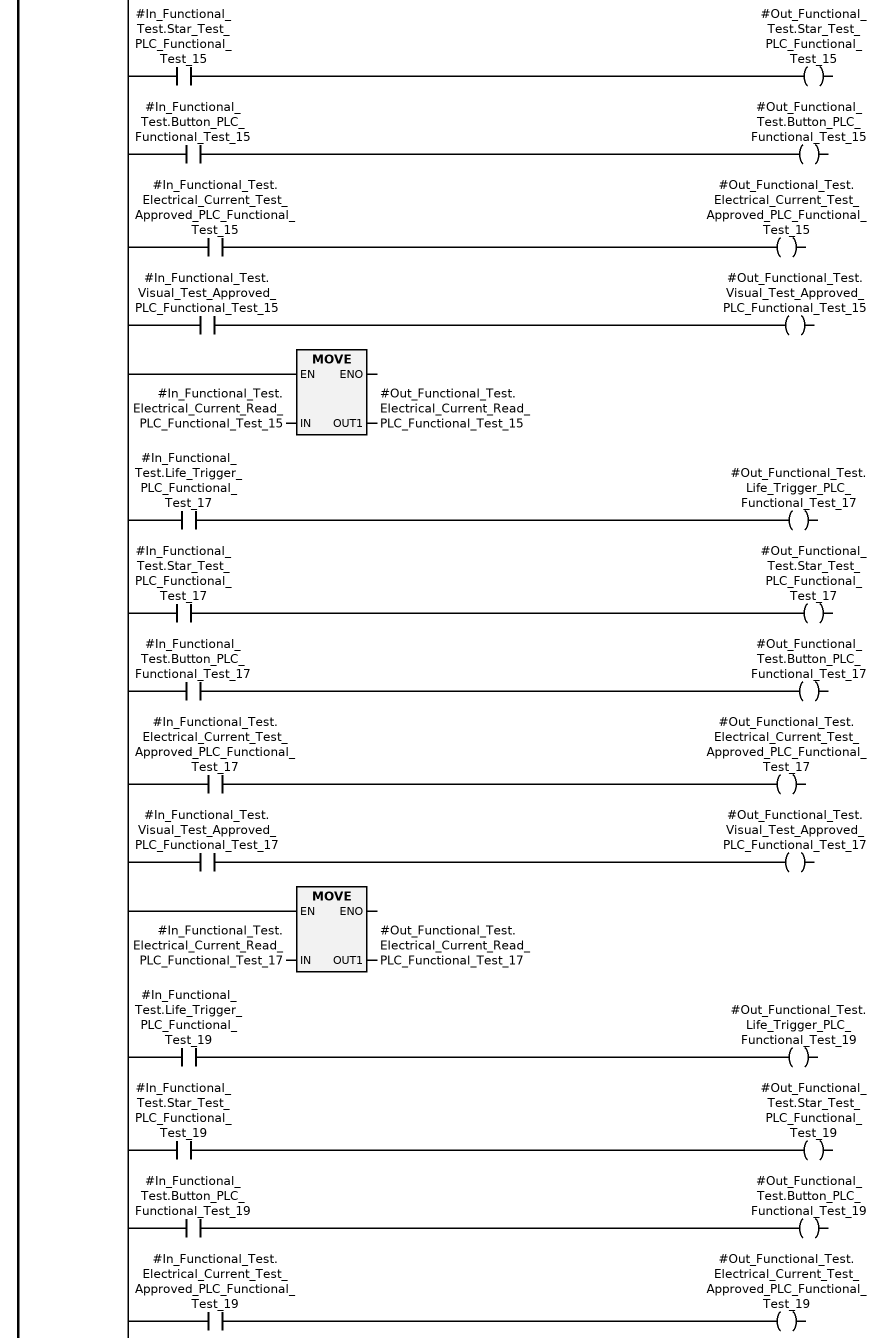
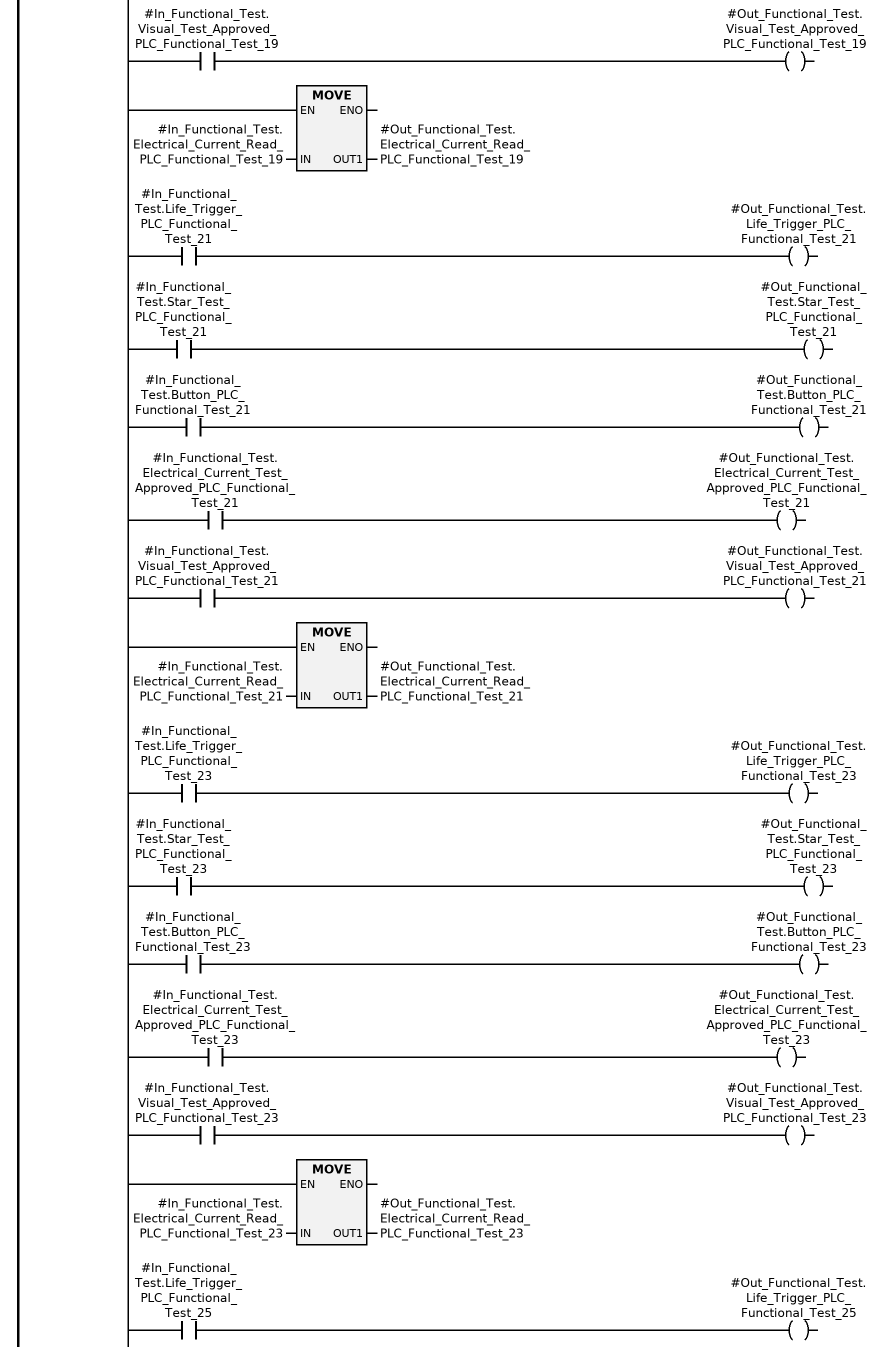
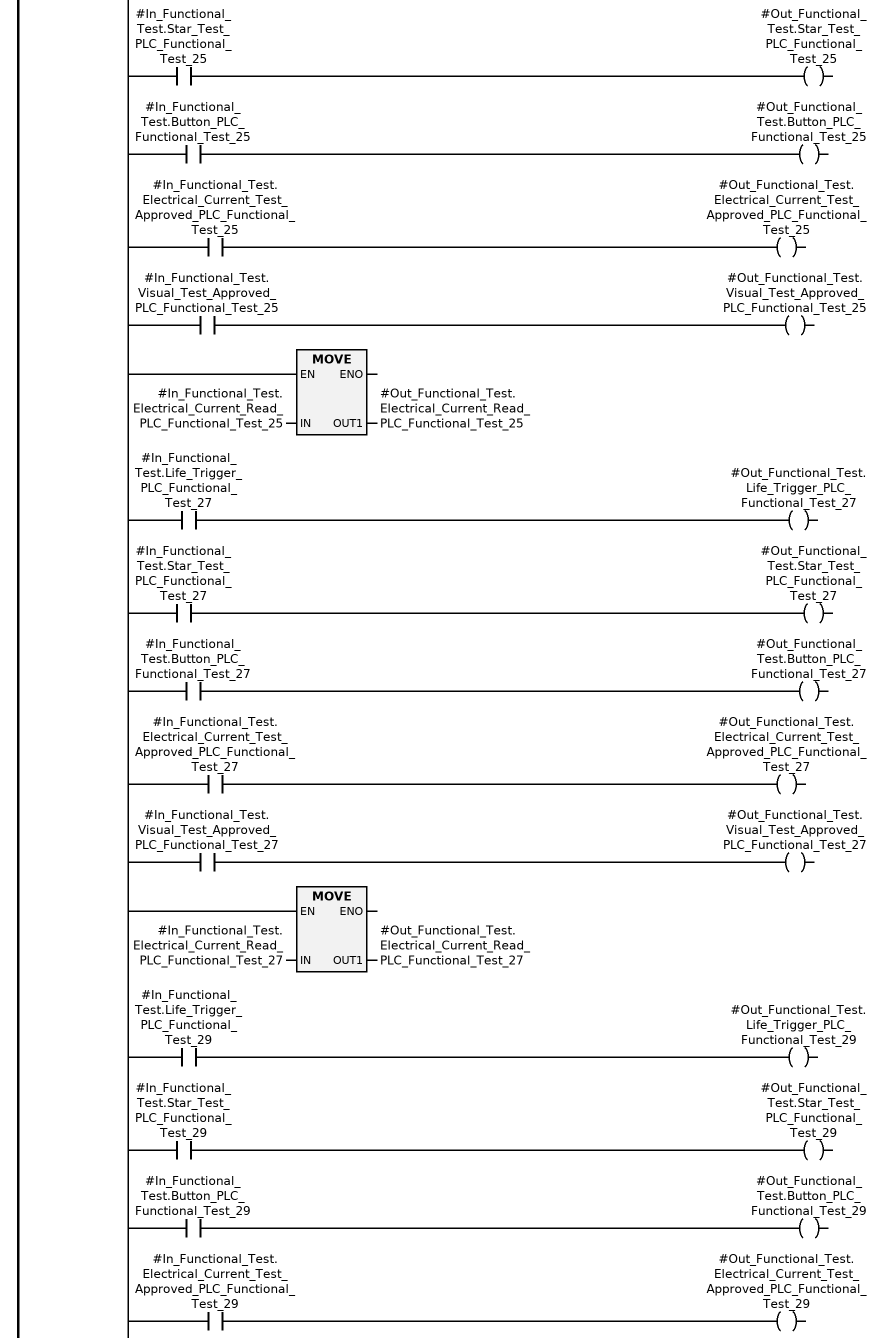
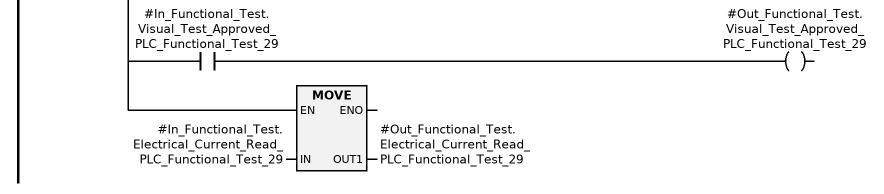
   RUNG wire#powerrail
      { S7_Templates := "SrcType := SInt" } EQ_Contact(in1 := #Test_Station, in2 := 1)
      wire#w1
      Contact( #Life_Trigger )
      Coil( #Out_Functional_Test.Life_Trigger_PLC_Functional_Test_1 )
   END_RUNG
   RUNG wire#w1
      Contact( #Star_Test )
      Coil( #Out_Functional_Test.Star_Test_PLC_Functional_Test_1 )
   END_RUNG
   RUNG wire#w1
      Contact( #Button_Start_Approve )
      Coil( #Out_Functional_Test.Button_PLC_Functional_Test_1 )
   END_RUNG
   RUNG wire#w1
      Contact( #Electrical_Current_Test_Approved )
      Coil( #Out_Functional_Test.Electrical_Current_Test_Approved_PLC_Functional_Test_1 )
   END_RUNG
   RUNG wire#w1
      Contact( #Visual_Test_Approved )
      Coil( #Out_Functional_Test.Visual_Test_Approved_PLC_Functional_Test_1 )
   END_RUNG
   RUNG wire#w1
      Contact( #In_Test_Parameters.Reset_PLC_Functional_Test_1 )
      Coil( #Reset_Functional_Test )
   END_RUNG
   RUNG wire#w1
      Move(in := #Electrical_Current_Read, out1 => #Out_Functional_Test.Electrical_Current_Read_PLC_Functional_Test_1)
      Move(in := #Electrical_Voltage_Read, out1 => #Out_Electrical_Voltage_Read)
   END_RUNG
   RUNG wire#w1
      Contact( #In_Functional_Test.Life_Trigger_PLC_Functional_Test_3 )
      Coil( #Out_Functional_Test.Life_Trigger_PLC_Functional_Test_3 )
   END_RUNG
   RUNG wire#w1
      Contact( #In_Functional_Test.Star_Test_PLC_Functional_Test_3 )
      Coil( #Out_Functional_Test.Star_Test_PLC_Functional_Test_3 )
   END_RUNG
   RUNG wire#w1
      Contact( #In_Functional_Test.Button_PLC_Functional_Test_3 )
      Coil( #Out_Functional_Test.Button_PLC_Functional_Test_3 )
   END_RUNG
   RUNG wire#w1
      Contact( #In_Functional_Test.Electrical_Current_Test_Approved_PLC_Functional_Test_3 )
      Coil( #Out_Functional_Test.Electrical_Current_Test_Approved_PLC_Functional_Test_3 )
   END_RUNG
   RUNG wire#w1
      Contact( #In_Functional_Test.Visual_Test_Approved_PLC_Functional_Test_3 )
      Coil( #Out_Functional_Test.Visual_Test_Approved_PLC_Functional_Test_3 )
   END_RUNG
   RUNG wire#w1
      Move(in := #In_Functional_Test.Electrical_Current_Read_PLC_Functional_Test_3, out1 => #Out_Functional_Test.Electrical_Current_Read_PLC_Functional_Test_3)
   END_RUNG
   RUNG wire#w1
      Contact( #In_Functional_Test.Life_Trigger_PLC_Functional_Test_5 )
      Coil( #Out_Functional_Test.Life_Trigger_PLC_Functional_Test_5 )
   END_RUNG
   RUNG wire#w1
      Contact( #In_Functional_Test.Star_Test_PLC_Functional_Test_5 )
      Coil( #Out_Functional_Test.Star_Test_PLC_Functional_Test_5 )
   END_RUNG
   RUNG wire#w1
      Contact( #In_Functional_Test.Button_PLC_Functional_Test_5 )
      Coil( #Out_Functional_Test.Button_PLC_Functional_Test_5 )
   END_RUNG
   RUNG wire#w1
      Contact( #In_Functional_Test.Electrical_Current_Test_Approved_PLC_Functional_Test_5 )
      Coil( #Out_Functional_Test.Electrical_Current_Test_Approved_PLC_Functional_Test_5 )
   END_RUNG
   RUNG wire#w1
      Contact( #In_Functional_Test.Visual_Test_Approved_PLC_Functional_Test_5 )
      Coil( #Out_Functional_Test.Visual_Test_Approved_PLC_Functional_Test_5 )
   END_RUNG
   RUNG wire#w1
      Move(in := #In_Functional_Test.Electrical_Current_Read_PLC_Functional_Test_5, out1 => #Out_Functional_Test.Electrical_Current_Read_PLC_Functional_Test_5)
   END_RUNG
   RUNG wire#w1
      Contact( #In_Functional_Test.Life_Trigger_PLC_Functional_Test_7 )
      Coil( #Out_Functional_Test.Life_Trigger_PLC_Functional_Test_7 )
   END_RUNG
   RUNG wire#w1
      Contact( #In_Functional_Test.Star_Test_PLC_Functional_Test_7 )
      Coil( #Out_Functional_Test.Star_Test_PLC_Functional_Test_7 )
   END_RUNG
   RUNG wire#w1
      Contact( #In_Functional_Test.Button_PLC_Functional_Test_7 )
      Coil( #Out_Functional_Test.Button_PLC_Functional_Test_7 )
   END_RUNG
   RUNG wire#w1
      Contact( #In_Functional_Test.Electrical_Current_Test_Approved_PLC_Functional_Test_7 )
      Coil( #Out_Functional_Test.Electrical_Current_Test_Approved_PLC_Functional_Test_7 )
   END_RUNG
   RUNG wire#w1
      Contact( #In_Functional_Test.Visual_Test_Approved_PLC_Functional_Test_7 )
      Coil( #Out_Functional_Test.Visual_Test_Approved_PLC_Functional_Test_7 )
   END_RUNG
   RUNG wire#w1
      Move(in := #In_Functional_Test.Electrical_Current_Read_PLC_Functional_Test_7, out1 => #Out_Functional_Test.Electrical_Current_Read_PLC_Functional_Test_7)
   END_RUNG
   RUNG wire#w1
      Contact( #In_Functional_Test.Life_Trigger_PLC_Functional_Test_9 )
      Coil( #Out_Functional_Test.Life_Trigger_PLC_Functional_Test_9 )
   END_RUNG
   RUNG wire#w1
      Contact( #In_Functional_Test.Star_Test_PLC_Functional_Test_9 )
      Coil( #Out_Functional_Test.Star_Test_PLC_Functional_Test_9 )
   END_RUNG
   RUNG wire#w1
      Contact( #In_Functional_Test.Button_PLC_Functional_Test_9 )
      Coil( #Out_Functional_Test.Button_PLC_Functional_Test_9 )
   END_RUNG
   RUNG wire#w1
      Contact( #In_Functional_Test.Electrical_Current_Test_Approved_PLC_Functional_Test_9 )
      Coil( #Out_Functional_Test.Electrical_Current_Test_Approved_PLC_Functional_Test_9 )
   END_RUNG
   RUNG wire#w1
      Contact( #In_Functional_Test.Visual_Test_Approved_PLC_Functional_Test_9 )
      Coil( #Out_Functional_Test.Visual_Test_Approved_PLC_Functional_Test_9 )
   END_RUNG
   RUNG wire#w1
      Move(in := #In_Functional_Test.Electrical_Current_Read_PLC_Functional_Test_9, out1 => #Out_Functional_Test.Electrical_Current_Read_PLC_Functional_Test_9)
   END_RUNG
   RUNG wire#w1
      Contact( #In_Functional_Test.Life_Trigger_PLC_Functional_Test_11 )
      Coil( #Out_Functional_Test.Life_Trigger_PLC_Functional_Test_11 )
   END_RUNG
   RUNG wire#w1
      Contact( #In_Functional_Test.Star_Test_PLC_Functional_Test_11 )
      Coil( #Out_Functional_Test.Star_Test_PLC_Functional_Test_11 )
   END_RUNG
   RUNG wire#w1
      Contact( #In_Functional_Test.Button_PLC_Functional_Test_11 )
      Coil( #Out_Functional_Test.Button_PLC_Functional_Test_11 )
   END_RUNG
   RUNG wire#w1
      Contact( #In_Functional_Test.Electrical_Current_Test_Approved_PLC_Functional_Test_11 )
      Coil( #Out_Functional_Test.Electrical_Current_Test_Approved_PLC_Functional_Test_11 )
   END_RUNG
   RUNG wire#w1
      Contact( #In_Functional_Test.Visual_Test_Approved_PLC_Functional_Test_11 )
      Coil( #Out_Functional_Test.Visual_Test_Approved_PLC_Functional_Test_11 )
   END_RUNG
   RUNG wire#w1
      Move(in := #In_Functional_Test.Electrical_Current_Read_PLC_Functional_Test_11, out1 => #Out_Functional_Test.Electrical_Current_Read_PLC_Functional_Test_11)
   END_RUNG
   RUNG wire#w1
      Contact( #In_Functional_Test.Life_Trigger_PLC_Functional_Test_13 )
      Coil( #Out_Functional_Test.Life_Trigger_PLC_Functional_Test_13 )
   END_RUNG
   RUNG wire#w1
      Contact( #In_Functional_Test.Star_Test_PLC_Functional_Test_13 )
      Coil( #Out_Functional_Test.Star_Test_PLC_Functional_Test_13 )
   END_RUNG
   RUNG wire#w1
      Contact( #In_Functional_Test.Button_PLC_Functional_Test_13 )
      Coil( #Out_Functional_Test.Button_PLC_Functional_Test_13 )
   END_RUNG
   RUNG wire#w1
      Contact( #In_Functional_Test.Electrical_Current_Test_Approved_PLC_Functional_Test_13 )
      Coil( #Out_Functional_Test.Electrical_Current_Test_Approved_PLC_Functional_Test_13 )
   END_RUNG
   RUNG wire#w1
      Contact( #In_Functional_Test.Visual_Test_Approved_PLC_Functional_Test_13 )
      Coil( #Out_Functional_Test.Visual_Test_Approved_PLC_Functional_Test_13 )
   END_RUNG
   RUNG wire#w1
      Move(in := #In_Functional_Test.Electrical_Current_Read_PLC_Functional_Test_13, out1 => #Out_Functional_Test.Electrical_Current_Read_PLC_Functional_Test_13)
   END_RUNG
   RUNG wire#w1
      Contact( #In_Functional_Test.Life_Trigger_PLC_Functional_Test_15 )
      Coil( #Out_Functional_Test.Life_Trigger_PLC_Functional_Test_15 )
   END_RUNG
   RUNG wire#w1
      Contact( #In_Functional_Test.Star_Test_PLC_Functional_Test_15 )
      Coil( #Out_Functional_Test.Star_Test_PLC_Functional_Test_15 )
   END_RUNG
   RUNG wire#w1
      Contact( #In_Functional_Test.Button_PLC_Functional_Test_15 )
      Coil( #Out_Functional_Test.Button_PLC_Functional_Test_15 )
   END_RUNG
   RUNG wire#w1
      Contact( #In_Functional_Test.Electrical_Current_Test_Approved_PLC_Functional_Test_15 )
      Coil( #Out_Functional_Test.Electrical_Current_Test_Approved_PLC_Functional_Test_15 )
   END_RUNG
   RUNG wire#w1
      Contact( #In_Functional_Test.Visual_Test_Approved_PLC_Functional_Test_15 )
      Coil( #Out_Functional_Test.Visual_Test_Approved_PLC_Functional_Test_15 )
   END_RUNG
   RUNG wire#w1
      Move(in := #In_Functional_Test.Electrical_Current_Read_PLC_Functional_Test_15, out1 => #Out_Functional_Test.Electrical_Current_Read_PLC_Functional_Test_15)
   END_RUNG
   RUNG wire#w1
      Contact( #In_Functional_Test.Life_Trigger_PLC_Functional_Test_17 )
      Coil( #Out_Functional_Test.Life_Trigger_PLC_Functional_Test_17 )
   END_RUNG
   RUNG wire#w1
      Contact( #In_Functional_Test.Star_Test_PLC_Functional_Test_17 )
      Coil( #Out_Functional_Test.Star_Test_PLC_Functional_Test_17 )
   END_RUNG
   RUNG wire#w1
      Contact( #In_Functional_Test.Button_PLC_Functional_Test_17 )
      Coil( #Out_Functional_Test.Button_PLC_Functional_Test_17 )
   END_RUNG
   RUNG wire#w1
      Contact( #In_Functional_Test.Electrical_Current_Test_Approved_PLC_Functional_Test_17 )
      Coil( #Out_Functional_Test.Electrical_Current_Test_Approved_PLC_Functional_Test_17 )
   END_RUNG
   RUNG wire#w1
      Contact( #In_Functional_Test.Visual_Test_Approved_PLC_Functional_Test_17 )
      Coil( #Out_Functional_Test.Visual_Test_Approved_PLC_Functional_Test_17 )
   END_RUNG
   RUNG wire#w1
      Move(in := #In_Functional_Test.Electrical_Current_Read_PLC_Functional_Test_17, out1 => #Out_Functional_Test.Electrical_Current_Read_PLC_Functional_Test_17)
   END_RUNG
   RUNG wire#w1
      Contact( #In_Functional_Test.Life_Trigger_PLC_Functional_Test_19 )
      Coil( #Out_Functional_Test.Life_Trigger_PLC_Functional_Test_19 )
   END_RUNG
   RUNG wire#w1
      Contact( #In_Functional_Test.Star_Test_PLC_Functional_Test_19 )
      Coil( #Out_Functional_Test.Star_Test_PLC_Functional_Test_19 )
   END_RUNG
   RUNG wire#w1
      Contact( #In_Functional_Test.Button_PLC_Functional_Test_19 )
      Coil( #Out_Functional_Test.Button_PLC_Functional_Test_19 )
   END_RUNG
   RUNG wire#w1
      Contact( #In_Functional_Test.Electrical_Current_Test_Approved_PLC_Functional_Test_19 )
      Coil( #Out_Functional_Test.Electrical_Current_Test_Approved_PLC_Functional_Test_19 )
   END_RUNG
   RUNG wire#w1
      Contact( #In_Functional_Test.Visual_Test_Approved_PLC_Functional_Test_19 )
      Coil( #Out_Functional_Test.Visual_Test_Approved_PLC_Functional_Test_19 )
   END_RUNG
   RUNG wire#w1
      Move(in := #In_Functional_Test.Electrical_Current_Read_PLC_Functional_Test_19, out1 => #Out_Functional_Test.Electrical_Current_Read_PLC_Functional_Test_19)
   END_RUNG
   RUNG wire#w1
      Contact( #In_Functional_Test.Life_Trigger_PLC_Functional_Test_21 )
      Coil( #Out_Functional_Test.Life_Trigger_PLC_Functional_Test_21 )
   END_RUNG
   RUNG wire#w1
      Contact( #In_Functional_Test.Star_Test_PLC_Functional_Test_21 )
      Coil( #Out_Functional_Test.Star_Test_PLC_Functional_Test_21 )
   END_RUNG
   RUNG wire#w1
      Contact( #In_Functional_Test.Button_PLC_Functional_Test_21 )
      Coil( #Out_Functional_Test.Button_PLC_Functional_Test_21 )
   END_RUNG
   RUNG wire#w1
      Contact( #In_Functional_Test.Electrical_Current_Test_Approved_PLC_Functional_Test_21 )
      Coil( #Out_Functional_Test.Electrical_Current_Test_Approved_PLC_Functional_Test_21 )
   END_RUNG
   RUNG wire#w1
      Contact( #In_Functional_Test.Visual_Test_Approved_PLC_Functional_Test_21 )
      Coil( #Out_Functional_Test.Visual_Test_Approved_PLC_Functional_Test_21 )
   END_RUNG
   RUNG wire#w1
      Move(in := #In_Functional_Test.Electrical_Current_Read_PLC_Functional_Test_21, out1 => #Out_Functional_Test.Electrical_Current_Read_PLC_Functional_Test_21)
   END_RUNG
   RUNG wire#w1
      Contact( #In_Functional_Test.Life_Trigger_PLC_Functional_Test_23 )
      Coil( #Out_Functional_Test.Life_Trigger_PLC_Functional_Test_23 )
   END_RUNG
   RUNG wire#w1
      Contact( #In_Functional_Test.Star_Test_PLC_Functional_Test_23 )
      Coil( #Out_Functional_Test.Star_Test_PLC_Functional_Test_23 )
   END_RUNG
   RUNG wire#w1
      Contact( #In_Functional_Test.Button_PLC_Functional_Test_23 )
      Coil( #Out_Functional_Test.Button_PLC_Functional_Test_23 )
   END_RUNG
   RUNG wire#w1
      Contact( #In_Functional_Test.Electrical_Current_Test_Approved_PLC_Functional_Test_23 )
      Coil( #Out_Functional_Test.Electrical_Current_Test_Approved_PLC_Functional_Test_23 )
   END_RUNG
   RUNG wire#w1
      Contact( #In_Functional_Test.Visual_Test_Approved_PLC_Functional_Test_23 )
      Coil( #Out_Functional_Test.Visual_Test_Approved_PLC_Functional_Test_23 )
   END_RUNG
   RUNG wire#w1
      Move(in := #In_Functional_Test.Electrical_Current_Read_PLC_Functional_Test_23, out1 => #Out_Functional_Test.Electrical_Current_Read_PLC_Functional_Test_23)
   END_RUNG
   RUNG wire#w1
      Contact( #In_Functional_Test.Life_Trigger_PLC_Functional_Test_25 )
      Coil( #Out_Functional_Test.Life_Trigger_PLC_Functional_Test_25 )
   END_RUNG
   RUNG wire#w1
      Contact( #In_Functional_Test.Star_Test_PLC_Functional_Test_25 )
      Coil( #Out_Functional_Test.Star_Test_PLC_Functional_Test_25 )
   END_RUNG
   RUNG wire#w1
      Contact( #In_Functional_Test.Button_PLC_Functional_Test_25 )
      Coil( #Out_Functional_Test.Button_PLC_Functional_Test_25 )
   END_RUNG
   RUNG wire#w1
      Contact( #In_Functional_Test.Electrical_Current_Test_Approved_PLC_Functional_Test_25 )
      Coil( #Out_Functional_Test.Electrical_Current_Test_Approved_PLC_Functional_Test_25 )
   END_RUNG
   RUNG wire#w1
      Contact( #In_Functional_Test.Visual_Test_Approved_PLC_Functional_Test_25 )
      Coil( #Out_Functional_Test.Visual_Test_Approved_PLC_Functional_Test_25 )
   END_RUNG
   RUNG wire#w1
      Move(in := #In_Functional_Test.Electrical_Current_Read_PLC_Functional_Test_25, out1 => #Out_Functional_Test.Electrical_Current_Read_PLC_Functional_Test_25)
   END_RUNG
   RUNG wire#w1
      Contact( #In_Functional_Test.Life_Trigger_PLC_Functional_Test_27 )
      Coil( #Out_Functional_Test.Life_Trigger_PLC_Functional_Test_27 )
   END_RUNG
   RUNG wire#w1
      Contact( #In_Functional_Test.Star_Test_PLC_Functional_Test_27 )
      Coil( #Out_Functional_Test.Star_Test_PLC_Functional_Test_27 )
   END_RUNG
   RUNG wire#w1
      Contact( #In_Functional_Test.Button_PLC_Functional_Test_27 )
      Coil( #Out_Functional_Test.Button_PLC_Functional_Test_27 )
   END_RUNG
   RUNG wire#w1
      Contact( #In_Functional_Test.Electrical_Current_Test_Approved_PLC_Functional_Test_27 )
      Coil( #Out_Functional_Test.Electrical_Current_Test_Approved_PLC_Functional_Test_27 )
   END_RUNG
   RUNG wire#w1
      Contact( #In_Functional_Test.Visual_Test_Approved_PLC_Functional_Test_27 )
      Coil( #Out_Functional_Test.Visual_Test_Approved_PLC_Functional_Test_27 )
   END_RUNG
   RUNG wire#w1
      Move(in := #In_Functional_Test.Electrical_Current_Read_PLC_Functional_Test_27, out1 => #Out_Functional_Test.Electrical_Current_Read_PLC_Functional_Test_27)
   END_RUNG
   RUNG wire#w1
      Contact( #In_Functional_Test.Life_Trigger_PLC_Functional_Test_29 )
      Coil( #Out_Functional_Test.Life_Trigger_PLC_Functional_Test_29 )
   END_RUNG
   RUNG wire#w1
      Contact( #In_Functional_Test.Star_Test_PLC_Functional_Test_29 )
      Coil( #Out_Functional_Test.Star_Test_PLC_Functional_Test_29 )
   END_RUNG
   RUNG wire#w1
      Contact( #In_Functional_Test.Button_PLC_Functional_Test_29 )
      Coil( #Out_Functional_Test.Button_PLC_Functional_Test_29 )
   END_RUNG
   RUNG wire#w1
      Contact( #In_Functional_Test.Electrical_Current_Test_Approved_PLC_Functional_Test_29 )
      Coil( #Out_Functional_Test.Electrical_Current_Test_Approved_PLC_Functional_Test_29 )
   END_RUNG
   RUNG wire#w1
      Contact( #In_Functional_Test.Visual_Test_Approved_PLC_Functional_Test_29 )
      Coil( #Out_Functional_Test.Visual_Test_Approved_PLC_Functional_Test_29 )
   END_RUNG
   RUNG wire#w1
      Move(in := #In_Functional_Test.Electrical_Current_Read_PLC_Functional_Test_29, out1 => #Out_Functional_Test.Electrical_Current_Read_PLC_Functional_Test_29)
   END_RUNG
   // the same network as SCL:
   #_w1 := #Test_Station = 1;
   #Out_Functional_Test.Life_Trigger_PLC_Functional_Test_1 := #_w1 AND #Life_Trigger;
   #Out_Functional_Test.Star_Test_PLC_Functional_Test_1 := #_w1 AND #Star_Test;
   #Out_Functional_Test.Button_PLC_Functional_Test_1 := #_w1 AND #Button_Start_Approve;
   #Out_Functional_Test.Electrical_Current_Test_Approved_PLC_Functional_Test_1 := #_w1 AND #Electrical_Current_Test_Approved;
   #Out_Functional_Test.Visual_Test_Approved_PLC_Functional_Test_1 := #_w1 AND #Visual_Test_Approved;
   #Reset_Functional_Test := #_w1 AND #In_Test_Parameters.Reset_PLC_Functional_Test_1;
   IF #_w1 THEN
       #Out_Functional_Test.Electrical_Current_Read_PLC_Functional_Test_1 := #Electrical_Current_Read;
       #Out_Electrical_Voltage_Read := #Electrical_Voltage_Read;
   END_IF;
   #Out_Functional_Test.Life_Trigger_PLC_Functional_Test_3 := #_w1 AND #In_Functional_Test.Life_Trigger_PLC_Functional_Test_3;
   #Out_Functional_Test.Star_Test_PLC_Functional_Test_3 := #_w1 AND #In_Functional_Test.Star_Test_PLC_Functional_Test_3;
   #Out_Functional_Test.Button_PLC_Functional_Test_3 := #_w1 AND #In_Functional_Test.Button_PLC_Functional_Test_3;
   #Out_Functional_Test.Electrical_Current_Test_Approved_PLC_Functional_Test_3 := #_w1 AND #In_Functional_Test.Electrical_Current_Test_Approved_PLC_Functional_Test_3;
   #Out_Functional_Test.Visual_Test_Approved_PLC_Functional_Test_3 := #_w1 AND #In_Functional_Test.Visual_Test_Approved_PLC_Functional_Test_3;
   IF #_w1 THEN
       #Out_Functional_Test.Electrical_Current_Read_PLC_Functional_Test_3 := #In_Functional_Test.Electrical_Current_Read_PLC_Functional_Test_3;
   END_IF;
   #Out_Functional_Test.Life_Trigger_PLC_Functional_Test_5 := #_w1 AND #In_Functional_Test.Life_Trigger_PLC_Functional_Test_5;
   #Out_Functional_Test.Star_Test_PLC_Functional_Test_5 := #_w1 AND #In_Functional_Test.Star_Test_PLC_Functional_Test_5;
   #Out_Functional_Test.Button_PLC_Functional_Test_5 := #_w1 AND #In_Functional_Test.Button_PLC_Functional_Test_5;
   #Out_Functional_Test.Electrical_Current_Test_Approved_PLC_Functional_Test_5 := #_w1 AND #In_Functional_Test.Electrical_Current_Test_Approved_PLC_Functional_Test_5;
   #Out_Functional_Test.Visual_Test_Approved_PLC_Functional_Test_5 := #_w1 AND #In_Functional_Test.Visual_Test_Approved_PLC_Functional_Test_5;
   IF #_w1 THEN
       #Out_Functional_Test.Electrical_Current_Read_PLC_Functional_Test_5 := #In_Functional_Test.Electrical_Current_Read_PLC_Functional_Test_5;
   END_IF;
   #Out_Functional_Test.Life_Trigger_PLC_Functional_Test_7 := #_w1 AND #In_Functional_Test.Life_Trigger_PLC_Functional_Test_7;
   #Out_Functional_Test.Star_Test_PLC_Functional_Test_7 := #_w1 AND #In_Functional_Test.Star_Test_PLC_Functional_Test_7;
   #Out_Functional_Test.Button_PLC_Functional_Test_7 := #_w1 AND #In_Functional_Test.Button_PLC_Functional_Test_7;
   #Out_Functional_Test.Electrical_Current_Test_Approved_PLC_Functional_Test_7 := #_w1 AND #In_Functional_Test.Electrical_Current_Test_Approved_PLC_Functional_Test_7;
   #Out_Functional_Test.Visual_Test_Approved_PLC_Functional_Test_7 := #_w1 AND #In_Functional_Test.Visual_Test_Approved_PLC_Functional_Test_7;
   IF #_w1 THEN
       #Out_Functional_Test.Electrical_Current_Read_PLC_Functional_Test_7 := #In_Functional_Test.Electrical_Current_Read_PLC_Functional_Test_7;
   END_IF;
   #Out_Functional_Test.Life_Trigger_PLC_Functional_Test_9 := #_w1 AND #In_Functional_Test.Life_Trigger_PLC_Functional_Test_9;
   #Out_Functional_Test.Star_Test_PLC_Functional_Test_9 := #_w1 AND #In_Functional_Test.Star_Test_PLC_Functional_Test_9;
   #Out_Functional_Test.Button_PLC_Functional_Test_9 := #_w1 AND #In_Functional_Test.Button_PLC_Functional_Test_9;
   #Out_Functional_Test.Electrical_Current_Test_Approved_PLC_Functional_Test_9 := #_w1 AND #In_Functional_Test.Electrical_Current_Test_Approved_PLC_Functional_Test_9;
   #Out_Functional_Test.Visual_Test_Approved_PLC_Functional_Test_9 := #_w1 AND #In_Functional_Test.Visual_Test_Approved_PLC_Functional_Test_9;
   IF #_w1 THEN
       #Out_Functional_Test.Electrical_Current_Read_PLC_Functional_Test_9 := #In_Functional_Test.Electrical_Current_Read_PLC_Functional_Test_9;
   END_IF;
   #Out_Functional_Test.Life_Trigger_PLC_Functional_Test_11 := #_w1 AND #In_Functional_Test.Life_Trigger_PLC_Functional_Test_11;
   #Out_Functional_Test.Star_Test_PLC_Functional_Test_11 := #_w1 AND #In_Functional_Test.Star_Test_PLC_Functional_Test_11;
   #Out_Functional_Test.Button_PLC_Functional_Test_11 := #_w1 AND #In_Functional_Test.Button_PLC_Functional_Test_11;
   #Out_Functional_Test.Electrical_Current_Test_Approved_PLC_Functional_Test_11 := #_w1 AND #In_Functional_Test.Electrical_Current_Test_Approved_PLC_Functional_Test_11;
   #Out_Functional_Test.Visual_Test_Approved_PLC_Functional_Test_11 := #_w1 AND #In_Functional_Test.Visual_Test_Approved_PLC_Functional_Test_11;
   IF #_w1 THEN
       #Out_Functional_Test.Electrical_Current_Read_PLC_Functional_Test_11 := #In_Functional_Test.Electrical_Current_Read_PLC_Functional_Test_11;
   END_IF;
   #Out_Functional_Test.Life_Trigger_PLC_Functional_Test_13 := #_w1 AND #In_Functional_Test.Life_Trigger_PLC_Functional_Test_13;
   #Out_Functional_Test.Star_Test_PLC_Functional_Test_13 := #_w1 AND #In_Functional_Test.Star_Test_PLC_Functional_Test_13;
   #Out_Functional_Test.Button_PLC_Functional_Test_13 := #_w1 AND #In_Functional_Test.Button_PLC_Functional_Test_13;
   #Out_Functional_Test.Electrical_Current_Test_Approved_PLC_Functional_Test_13 := #_w1 AND #In_Functional_Test.Electrical_Current_Test_Approved_PLC_Functional_Test_13;
   #Out_Functional_Test.Visual_Test_Approved_PLC_Functional_Test_13 := #_w1 AND #In_Functional_Test.Visual_Test_Approved_PLC_Functional_Test_13;
   IF #_w1 THEN
       #Out_Functional_Test.Electrical_Current_Read_PLC_Functional_Test_13 := #In_Functional_Test.Electrical_Current_Read_PLC_Functional_Test_13;
   END_IF;
   #Out_Functional_Test.Life_Trigger_PLC_Functional_Test_15 := #_w1 AND #In_Functional_Test.Life_Trigger_PLC_Functional_Test_15;
   #Out_Functional_Test.Star_Test_PLC_Functional_Test_15 := #_w1 AND #In_Functional_Test.Star_Test_PLC_Functional_Test_15;
   #Out_Functional_Test.Button_PLC_Functional_Test_15 := #_w1 AND #In_Functional_Test.Button_PLC_Functional_Test_15;
   #Out_Functional_Test.Electrical_Current_Test_Approved_PLC_Functional_Test_15 := #_w1 AND #In_Functional_Test.Electrical_Current_Test_Approved_PLC_Functional_Test_15;
   #Out_Functional_Test.Visual_Test_Approved_PLC_Functional_Test_15 := #_w1 AND #In_Functional_Test.Visual_Test_Approved_PLC_Functional_Test_15;
   IF #_w1 THEN
       #Out_Functional_Test.Electrical_Current_Read_PLC_Functional_Test_15 := #In_Functional_Test.Electrical_Current_Read_PLC_Functional_Test_15;
   END_IF;
   #Out_Functional_Test.Life_Trigger_PLC_Functional_Test_17 := #_w1 AND #In_Functional_Test.Life_Trigger_PLC_Functional_Test_17;
   #Out_Functional_Test.Star_Test_PLC_Functional_Test_17 := #_w1 AND #In_Functional_Test.Star_Test_PLC_Functional_Test_17;
   #Out_Functional_Test.Button_PLC_Functional_Test_17 := #_w1 AND #In_Functional_Test.Button_PLC_Functional_Test_17;
   #Out_Functional_Test.Electrical_Current_Test_Approved_PLC_Functional_Test_17 := #_w1 AND #In_Functional_Test.Electrical_Current_Test_Approved_PLC_Functional_Test_17;
   #Out_Functional_Test.Visual_Test_Approved_PLC_Functional_Test_17 := #_w1 AND #In_Functional_Test.Visual_Test_Approved_PLC_Functional_Test_17;
   IF #_w1 THEN
       #Out_Functional_Test.Electrical_Current_Read_PLC_Functional_Test_17 := #In_Functional_Test.Electrical_Current_Read_PLC_Functional_Test_17;
   END_IF;
   #Out_Functional_Test.Life_Trigger_PLC_Functional_Test_19 := #_w1 AND #In_Functional_Test.Life_Trigger_PLC_Functional_Test_19;
   #Out_Functional_Test.Star_Test_PLC_Functional_Test_19 := #_w1 AND #In_Functional_Test.Star_Test_PLC_Functional_Test_19;
   #Out_Functional_Test.Button_PLC_Functional_Test_19 := #_w1 AND #In_Functional_Test.Button_PLC_Functional_Test_19;
   #Out_Functional_Test.Electrical_Current_Test_Approved_PLC_Functional_Test_19 := #_w1 AND #In_Functional_Test.Electrical_Current_Test_Approved_PLC_Functional_Test_19;
   #Out_Functional_Test.Visual_Test_Approved_PLC_Functional_Test_19 := #_w1 AND #In_Functional_Test.Visual_Test_Approved_PLC_Functional_Test_19;
   IF #_w1 THEN
       #Out_Functional_Test.Electrical_Current_Read_PLC_Functional_Test_19 := #In_Functional_Test.Electrical_Current_Read_PLC_Functional_Test_19;
   END_IF;
   #Out_Functional_Test.Life_Trigger_PLC_Functional_Test_21 := #_w1 AND #In_Functional_Test.Life_Trigger_PLC_Functional_Test_21;
   #Out_Functional_Test.Star_Test_PLC_Functional_Test_21 := #_w1 AND #In_Functional_Test.Star_Test_PLC_Functional_Test_21;
   #Out_Functional_Test.Button_PLC_Functional_Test_21 := #_w1 AND #In_Functional_Test.Button_PLC_Functional_Test_21;
   #Out_Functional_Test.Electrical_Current_Test_Approved_PLC_Functional_Test_21 := #_w1 AND #In_Functional_Test.Electrical_Current_Test_Approved_PLC_Functional_Test_21;
   #Out_Functional_Test.Visual_Test_Approved_PLC_Functional_Test_21 := #_w1 AND #In_Functional_Test.Visual_Test_Approved_PLC_Functional_Test_21;
   IF #_w1 THEN
       #Out_Functional_Test.Electrical_Current_Read_PLC_Functional_Test_21 := #In_Functional_Test.Electrical_Current_Read_PLC_Functional_Test_21;
   END_IF;
   #Out_Functional_Test.Life_Trigger_PLC_Functional_Test_23 := #_w1 AND #In_Functional_Test.Life_Trigger_PLC_Functional_Test_23;
   #Out_Functional_Test.Star_Test_PLC_Functional_Test_23 := #_w1 AND #In_Functional_Test.Star_Test_PLC_Functional_Test_23;
   #Out_Functional_Test.Button_PLC_Functional_Test_23 := #_w1 AND #In_Functional_Test.Button_PLC_Functional_Test_23;
   #Out_Functional_Test.Electrical_Current_Test_Approved_PLC_Functional_Test_23 := #_w1 AND #In_Functional_Test.Electrical_Current_Test_Approved_PLC_Functional_Test_23;
   #Out_Functional_Test.Visual_Test_Approved_PLC_Functional_Test_23 := #_w1 AND #In_Functional_Test.Visual_Test_Approved_PLC_Functional_Test_23;
   IF #_w1 THEN
       #Out_Functional_Test.Electrical_Current_Read_PLC_Functional_Test_23 := #In_Functional_Test.Electrical_Current_Read_PLC_Functional_Test_23;
   END_IF;
   #Out_Functional_Test.Life_Trigger_PLC_Functional_Test_25 := #_w1 AND #In_Functional_Test.Life_Trigger_PLC_Functional_Test_25;
   #Out_Functional_Test.Star_Test_PLC_Functional_Test_25 := #_w1 AND #In_Functional_Test.Star_Test_PLC_Functional_Test_25;
   #Out_Functional_Test.Button_PLC_Functional_Test_25 := #_w1 AND #In_Functional_Test.Button_PLC_Functional_Test_25;
   #Out_Functional_Test.Electrical_Current_Test_Approved_PLC_Functional_Test_25 := #_w1 AND #In_Functional_Test.Electrical_Current_Test_Approved_PLC_Functional_Test_25;
   #Out_Functional_Test.Visual_Test_Approved_PLC_Functional_Test_25 := #_w1 AND #In_Functional_Test.Visual_Test_Approved_PLC_Functional_Test_25;
   IF #_w1 THEN
       #Out_Functional_Test.Electrical_Current_Read_PLC_Functional_Test_25 := #In_Functional_Test.Electrical_Current_Read_PLC_Functional_Test_25;
   END_IF;
   #Out_Functional_Test.Life_Trigger_PLC_Functional_Test_27 := #_w1 AND #In_Functional_Test.Life_Trigger_PLC_Functional_Test_27;
   #Out_Functional_Test.Star_Test_PLC_Functional_Test_27 := #_w1 AND #In_Functional_Test.Star_Test_PLC_Functional_Test_27;
   #Out_Functional_Test.Button_PLC_Functional_Test_27 := #_w1 AND #In_Functional_Test.Button_PLC_Functional_Test_27;
   #Out_Functional_Test.Electrical_Current_Test_Approved_PLC_Functional_Test_27 := #_w1 AND #In_Functional_Test.Electrical_Current_Test_Approved_PLC_Functional_Test_27;
   #Out_Functional_Test.Visual_Test_Approved_PLC_Functional_Test_27 := #_w1 AND #In_Functional_Test.Visual_Test_Approved_PLC_Functional_Test_27;
   IF #_w1 THEN
       #Out_Functional_Test.Electrical_Current_Read_PLC_Functional_Test_27 := #In_Functional_Test.Electrical_Current_Read_PLC_Functional_Test_27;
   END_IF;
   #Out_Functional_Test.Life_Trigger_PLC_Functional_Test_29 := #_w1 AND #In_Functional_Test.Life_Trigger_PLC_Functional_Test_29;
   #Out_Functional_Test.Star_Test_PLC_Functional_Test_29 := #_w1 AND #In_Functional_Test.Star_Test_PLC_Functional_Test_29;
   #Out_Functional_Test.Button_PLC_Functional_Test_29 := #_w1 AND #In_Functional_Test.Button_PLC_Functional_Test_29;
   #Out_Functional_Test.Electrical_Current_Test_Approved_PLC_Functional_Test_29 := #_w1 AND #In_Functional_Test.Electrical_Current_Test_Approved_PLC_Functional_Test_29;
   #Out_Functional_Test.Visual_Test_Approved_PLC_Functional_Test_29 := #_w1 AND #In_Functional_Test.Visual_Test_Approved_PLC_Functional_Test_29;
   IF #_w1 THEN
       #Out_Functional_Test.Electrical_Current_Read_PLC_Functional_Test_29 := #In_Functional_Test.Electrical_Current_Read_PLC_Functional_Test_29;
   END_IF;
END_REGION

REGION Network 3: Functional Test Station 3
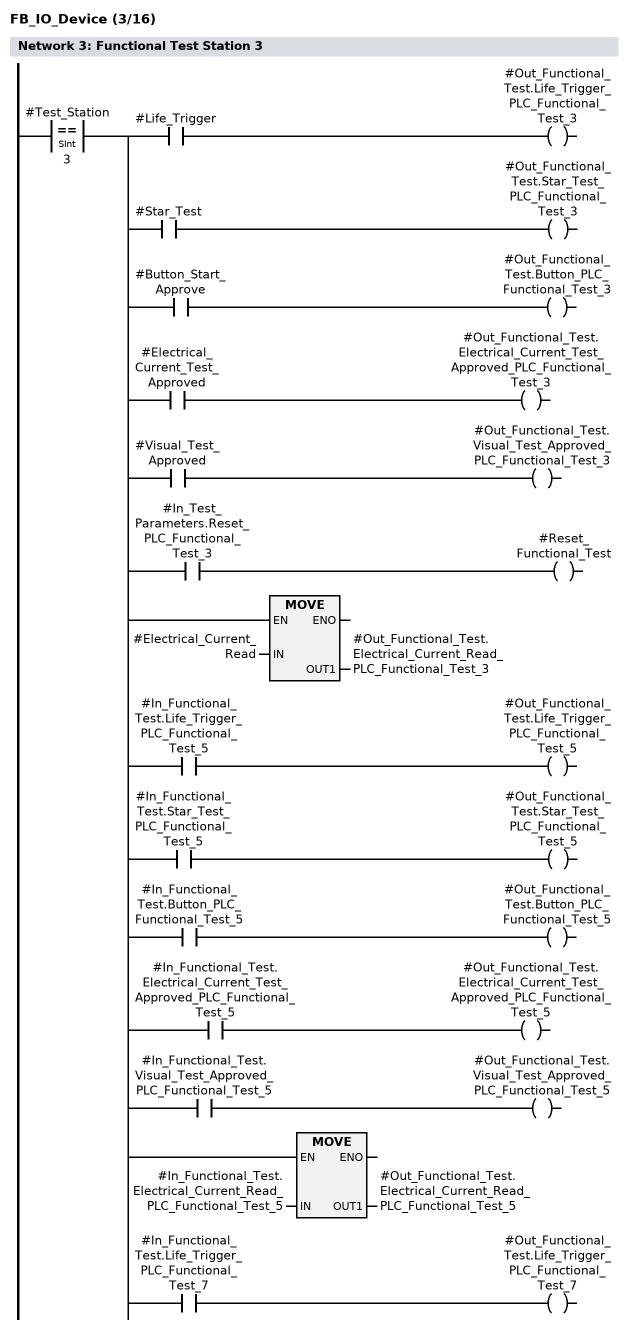
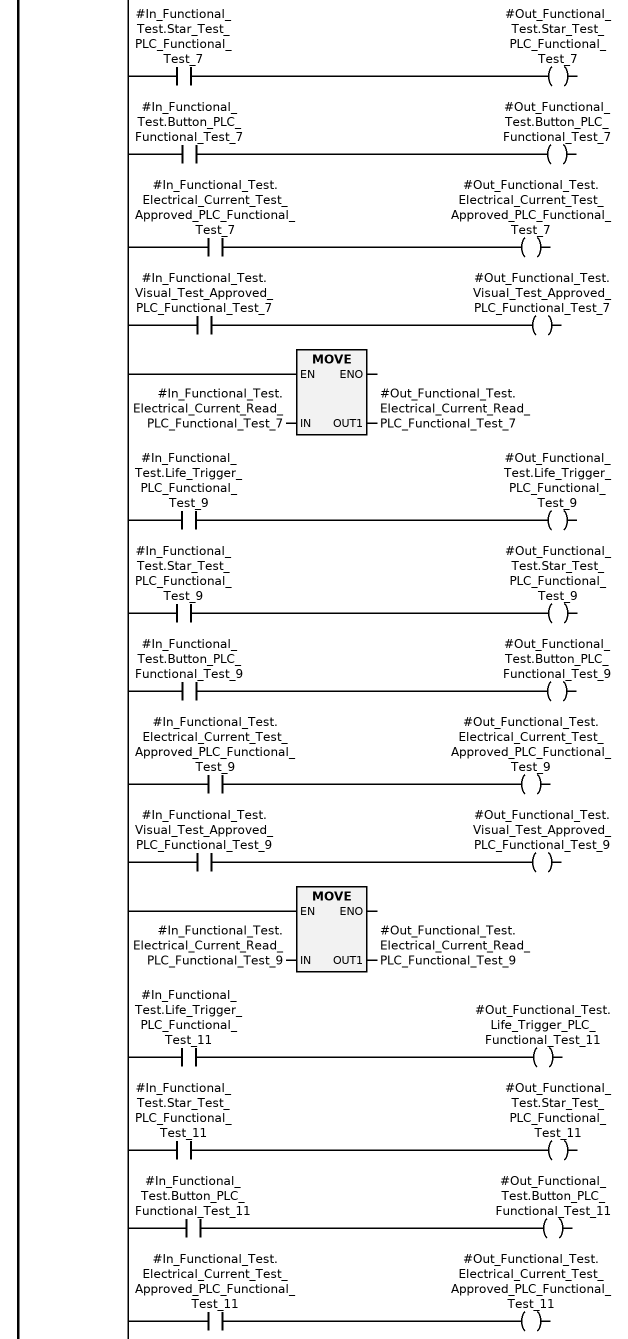
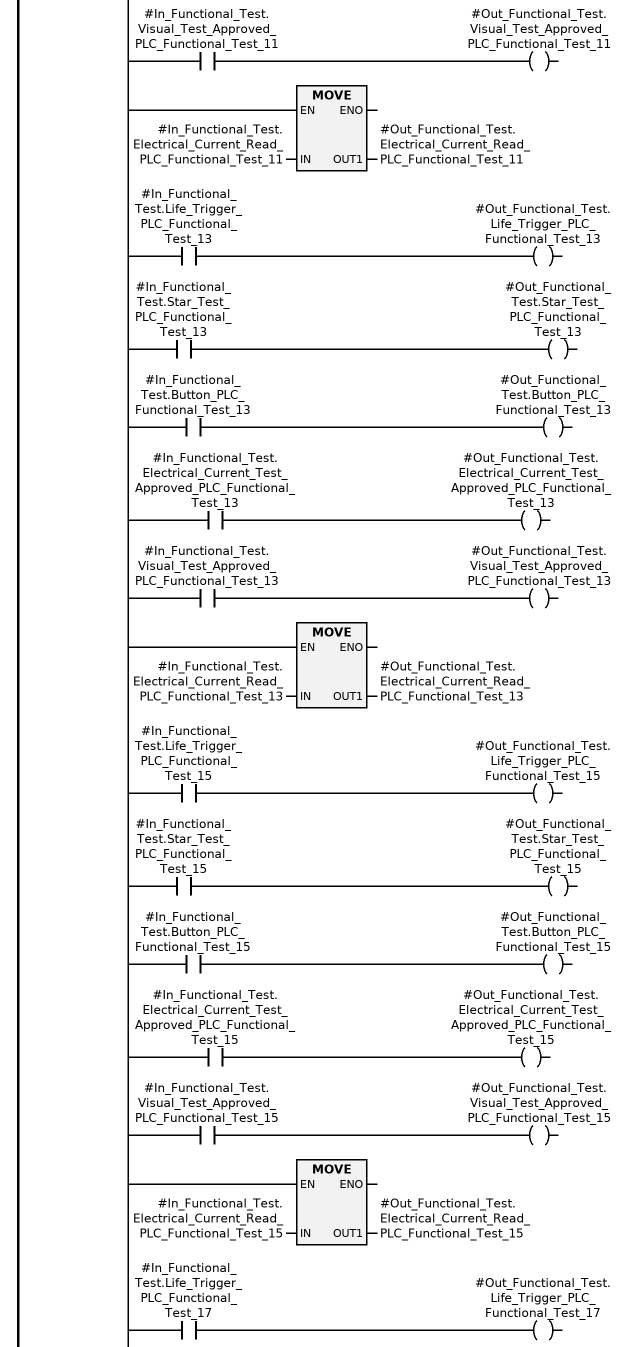
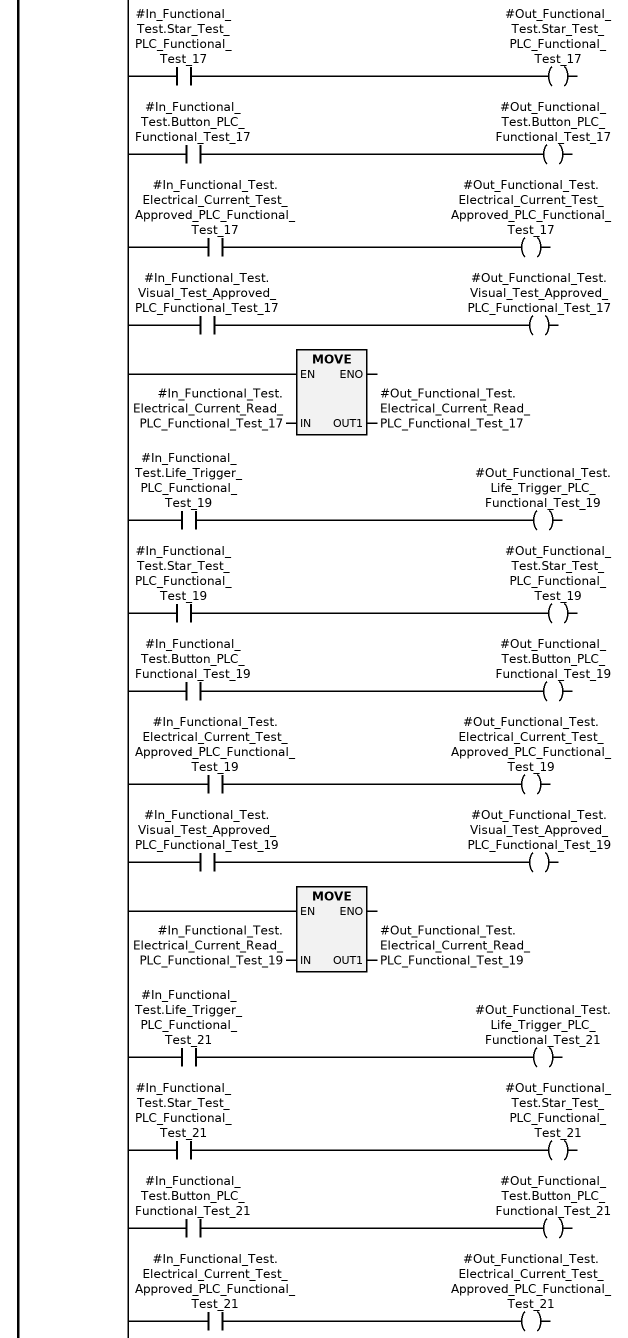
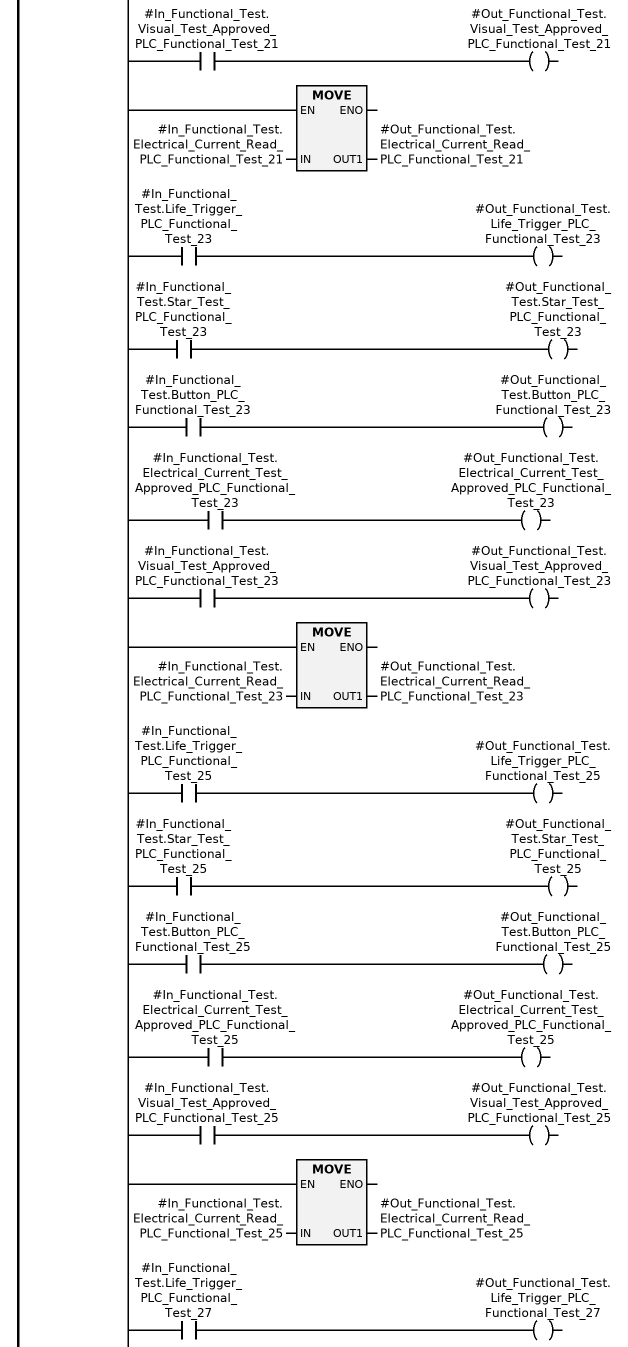
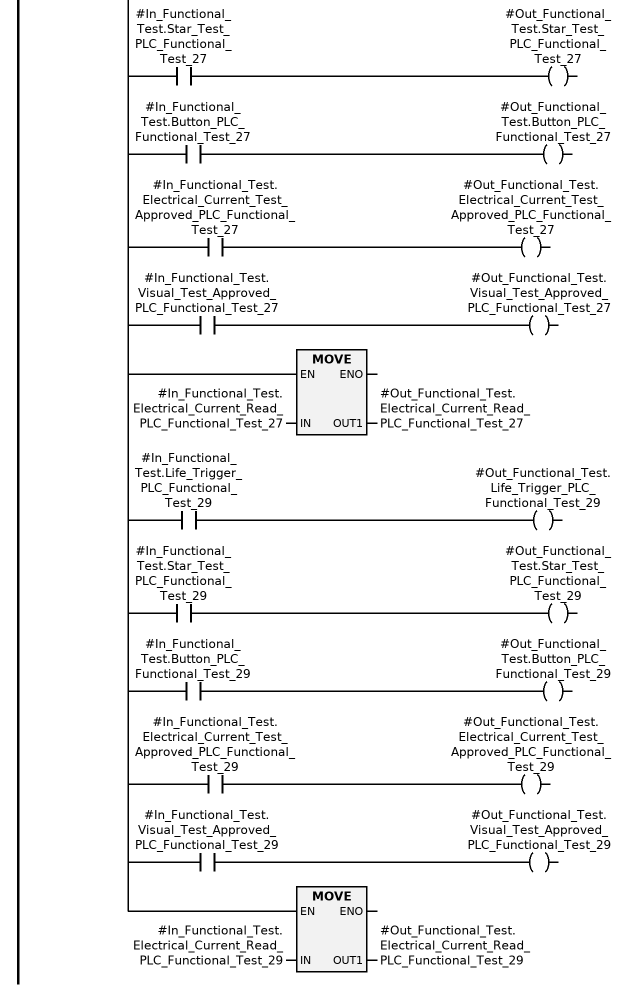
   RUNG wire#powerrail
      { S7_Templates := "SrcType := SInt" } EQ_Contact(in1 := #Test_Station, in2 := 3)
      wire#w1
      Contact( #Life_Trigger )
      Coil( #Out_Functional_Test.Life_Trigger_PLC_Functional_Test_3 )
   END_RUNG
   RUNG wire#w1
      Contact( #Star_Test )
      Coil( #Out_Functional_Test.Star_Test_PLC_Functional_Test_3 )
   END_RUNG
   RUNG wire#w1
      Contact( #Button_Start_Approve )
      Coil( #Out_Functional_Test.Button_PLC_Functional_Test_3 )
   END_RUNG
   RUNG wire#w1
      Contact( #Electrical_Current_Test_Approved )
      Coil( #Out_Functional_Test.Electrical_Current_Test_Approved_PLC_Functional_Test_3 )
   END_RUNG
   RUNG wire#w1
      Contact( #Visual_Test_Approved )
      Coil( #Out_Functional_Test.Visual_Test_Approved_PLC_Functional_Test_3 )
   END_RUNG
   RUNG wire#w1
      Contact( #In_Test_Parameters.Reset_PLC_Functional_Test_3 )
      Coil( #Reset_Functional_Test )
   END_RUNG
   RUNG wire#w1
      Move(in := #Electrical_Current_Read, out1 => #Out_Functional_Test.Electrical_Current_Read_PLC_Functional_Test_3)
   END_RUNG
   RUNG wire#w1
      Contact( #In_Functional_Test.Life_Trigger_PLC_Functional_Test_5 )
      Coil( #Out_Functional_Test.Life_Trigger_PLC_Functional_Test_5 )
   END_RUNG
   RUNG wire#w1
      Contact( #In_Functional_Test.Star_Test_PLC_Functional_Test_5 )
      Coil( #Out_Functional_Test.Star_Test_PLC_Functional_Test_5 )
   END_RUNG
   RUNG wire#w1
      Contact( #In_Functional_Test.Button_PLC_Functional_Test_5 )
      Coil( #Out_Functional_Test.Button_PLC_Functional_Test_5 )
   END_RUNG
   RUNG wire#w1
      Contact( #In_Functional_Test.Electrical_Current_Test_Approved_PLC_Functional_Test_5 )
      Coil( #Out_Functional_Test.Electrical_Current_Test_Approved_PLC_Functional_Test_5 )
   END_RUNG
   RUNG wire#w1
      Contact( #In_Functional_Test.Visual_Test_Approved_PLC_Functional_Test_5 )
      Coil( #Out_Functional_Test.Visual_Test_Approved_PLC_Functional_Test_5 )
   END_RUNG
   RUNG wire#w1
      Move(in := #In_Functional_Test.Electrical_Current_Read_PLC_Functional_Test_5, out1 => #Out_Functional_Test.Electrical_Current_Read_PLC_Functional_Test_5)
   END_RUNG
   RUNG wire#w1
      Contact( #In_Functional_Test.Life_Trigger_PLC_Functional_Test_7 )
      Coil( #Out_Functional_Test.Life_Trigger_PLC_Functional_Test_7 )
   END_RUNG
   RUNG wire#w1
      Contact( #In_Functional_Test.Star_Test_PLC_Functional_Test_7 )
      Coil( #Out_Functional_Test.Star_Test_PLC_Functional_Test_7 )
   END_RUNG
   RUNG wire#w1
      Contact( #In_Functional_Test.Button_PLC_Functional_Test_7 )
      Coil( #Out_Functional_Test.Button_PLC_Functional_Test_7 )
   END_RUNG
   RUNG wire#w1
      Contact( #In_Functional_Test.Electrical_Current_Test_Approved_PLC_Functional_Test_7 )
      Coil( #Out_Functional_Test.Electrical_Current_Test_Approved_PLC_Functional_Test_7 )
   END_RUNG
   RUNG wire#w1
      Contact( #In_Functional_Test.Visual_Test_Approved_PLC_Functional_Test_7 )
      Coil( #Out_Functional_Test.Visual_Test_Approved_PLC_Functional_Test_7 )
   END_RUNG
   RUNG wire#w1
      Move(in := #In_Functional_Test.Electrical_Current_Read_PLC_Functional_Test_7, out1 => #Out_Functional_Test.Electrical_Current_Read_PLC_Functional_Test_7)
   END_RUNG
   RUNG wire#w1
      Contact( #In_Functional_Test.Life_Trigger_PLC_Functional_Test_9 )
      Coil( #Out_Functional_Test.Life_Trigger_PLC_Functional_Test_9 )
   END_RUNG
   RUNG wire#w1
      Contact( #In_Functional_Test.Star_Test_PLC_Functional_Test_9 )
      Coil( #Out_Functional_Test.Star_Test_PLC_Functional_Test_9 )
   END_RUNG
   RUNG wire#w1
      Contact( #In_Functional_Test.Button_PLC_Functional_Test_9 )
      Coil( #Out_Functional_Test.Button_PLC_Functional_Test_9 )
   END_RUNG
   RUNG wire#w1
      Contact( #In_Functional_Test.Electrical_Current_Test_Approved_PLC_Functional_Test_9 )
      Coil( #Out_Functional_Test.Electrical_Current_Test_Approved_PLC_Functional_Test_9 )
   END_RUNG
   RUNG wire#w1
      Contact( #In_Functional_Test.Visual_Test_Approved_PLC_Functional_Test_9 )
      Coil( #Out_Functional_Test.Visual_Test_Approved_PLC_Functional_Test_9 )
   END_RUNG
   RUNG wire#w1
      Move(in := #In_Functional_Test.Electrical_Current_Read_PLC_Functional_Test_9, out1 => #Out_Functional_Test.Electrical_Current_Read_PLC_Functional_Test_9)
   END_RUNG
   RUNG wire#w1
      Contact( #In_Functional_Test.Life_Trigger_PLC_Functional_Test_11 )
      Coil( #Out_Functional_Test.Life_Trigger_PLC_Functional_Test_11 )
   END_RUNG
   RUNG wire#w1
      Contact( #In_Functional_Test.Star_Test_PLC_Functional_Test_11 )
      Coil( #Out_Functional_Test.Star_Test_PLC_Functional_Test_11 )
   END_RUNG
   RUNG wire#w1
      Contact( #In_Functional_Test.Button_PLC_Functional_Test_11 )
      Coil( #Out_Functional_Test.Button_PLC_Functional_Test_11 )
   END_RUNG
   RUNG wire#w1
      Contact( #In_Functional_Test.Electrical_Current_Test_Approved_PLC_Functional_Test_11 )
      Coil( #Out_Functional_Test.Electrical_Current_Test_Approved_PLC_Functional_Test_11 )
   END_RUNG
   RUNG wire#w1
      Contact( #In_Functional_Test.Visual_Test_Approved_PLC_Functional_Test_11 )
      Coil( #Out_Functional_Test.Visual_Test_Approved_PLC_Functional_Test_11 )
   END_RUNG
   RUNG wire#w1
      Move(in := #In_Functional_Test.Electrical_Current_Read_PLC_Functional_Test_11, out1 => #Out_Functional_Test.Electrical_Current_Read_PLC_Functional_Test_11)
   END_RUNG
   RUNG wire#w1
      Contact( #In_Functional_Test.Life_Trigger_PLC_Functional_Test_13 )
      Coil( #Out_Functional_Test.Life_Trigger_PLC_Functional_Test_13 )
   END_RUNG
   RUNG wire#w1
      Contact( #In_Functional_Test.Star_Test_PLC_Functional_Test_13 )
      Coil( #Out_Functional_Test.Star_Test_PLC_Functional_Test_13 )
   END_RUNG
   RUNG wire#w1
      Contact( #In_Functional_Test.Button_PLC_Functional_Test_13 )
      Coil( #Out_Functional_Test.Button_PLC_Functional_Test_13 )
   END_RUNG
   RUNG wire#w1
      Contact( #In_Functional_Test.Electrical_Current_Test_Approved_PLC_Functional_Test_13 )
      Coil( #Out_Functional_Test.Electrical_Current_Test_Approved_PLC_Functional_Test_13 )
   END_RUNG
   RUNG wire#w1
      Contact( #In_Functional_Test.Visual_Test_Approved_PLC_Functional_Test_13 )
      Coil( #Out_Functional_Test.Visual_Test_Approved_PLC_Functional_Test_13 )
   END_RUNG
   RUNG wire#w1
      Move(in := #In_Functional_Test.Electrical_Current_Read_PLC_Functional_Test_13, out1 => #Out_Functional_Test.Electrical_Current_Read_PLC_Functional_Test_13)
   END_RUNG
   RUNG wire#w1
      Contact( #In_Functional_Test.Life_Trigger_PLC_Functional_Test_15 )
      Coil( #Out_Functional_Test.Life_Trigger_PLC_Functional_Test_15 )
   END_RUNG
   RUNG wire#w1
      Contact( #In_Functional_Test.Star_Test_PLC_Functional_Test_15 )
      Coil( #Out_Functional_Test.Star_Test_PLC_Functional_Test_15 )
   END_RUNG
   RUNG wire#w1
      Contact( #In_Functional_Test.Button_PLC_Functional_Test_15 )
      Coil( #Out_Functional_Test.Button_PLC_Functional_Test_15 )
   END_RUNG
   RUNG wire#w1
      Contact( #In_Functional_Test.Electrical_Current_Test_Approved_PLC_Functional_Test_15 )
      Coil( #Out_Functional_Test.Electrical_Current_Test_Approved_PLC_Functional_Test_15 )
   END_RUNG
   RUNG wire#w1
      Contact( #In_Functional_Test.Visual_Test_Approved_PLC_Functional_Test_15 )
      Coil( #Out_Functional_Test.Visual_Test_Approved_PLC_Functional_Test_15 )
   END_RUNG
   RUNG wire#w1
      Move(in := #In_Functional_Test.Electrical_Current_Read_PLC_Functional_Test_15, out1 => #Out_Functional_Test.Electrical_Current_Read_PLC_Functional_Test_15)
   END_RUNG
   RUNG wire#w1
      Contact( #In_Functional_Test.Life_Trigger_PLC_Functional_Test_17 )
      Coil( #Out_Functional_Test.Life_Trigger_PLC_Functional_Test_17 )
   END_RUNG
   RUNG wire#w1
      Contact( #In_Functional_Test.Star_Test_PLC_Functional_Test_17 )
      Coil( #Out_Functional_Test.Star_Test_PLC_Functional_Test_17 )
   END_RUNG
   RUNG wire#w1
      Contact( #In_Functional_Test.Button_PLC_Functional_Test_17 )
      Coil( #Out_Functional_Test.Button_PLC_Functional_Test_17 )
   END_RUNG
   RUNG wire#w1
      Contact( #In_Functional_Test.Electrical_Current_Test_Approved_PLC_Functional_Test_17 )
      Coil( #Out_Functional_Test.Electrical_Current_Test_Approved_PLC_Functional_Test_17 )
   END_RUNG
   RUNG wire#w1
      Contact( #In_Functional_Test.Visual_Test_Approved_PLC_Functional_Test_17 )
      Coil( #Out_Functional_Test.Visual_Test_Approved_PLC_Functional_Test_17 )
   END_RUNG
   RUNG wire#w1
      Move(in := #In_Functional_Test.Electrical_Current_Read_PLC_Functional_Test_17, out1 => #Out_Functional_Test.Electrical_Current_Read_PLC_Functional_Test_17)
   END_RUNG
   RUNG wire#w1
      Contact( #In_Functional_Test.Life_Trigger_PLC_Functional_Test_19 )
      Coil( #Out_Functional_Test.Life_Trigger_PLC_Functional_Test_19 )
   END_RUNG
   RUNG wire#w1
      Contact( #In_Functional_Test.Star_Test_PLC_Functional_Test_19 )
      Coil( #Out_Functional_Test.Star_Test_PLC_Functional_Test_19 )
   END_RUNG
   RUNG wire#w1
      Contact( #In_Functional_Test.Button_PLC_Functional_Test_19 )
      Coil( #Out_Functional_Test.Button_PLC_Functional_Test_19 )
   END_RUNG
   RUNG wire#w1
      Contact( #In_Functional_Test.Electrical_Current_Test_Approved_PLC_Functional_Test_19 )
      Coil( #Out_Functional_Test.Electrical_Current_Test_Approved_PLC_Functional_Test_19 )
   END_RUNG
   RUNG wire#w1
      Contact( #In_Functional_Test.Visual_Test_Approved_PLC_Functional_Test_19 )
      Coil( #Out_Functional_Test.Visual_Test_Approved_PLC_Functional_Test_19 )
   END_RUNG
   RUNG wire#w1
      Move(in := #In_Functional_Test.Electrical_Current_Read_PLC_Functional_Test_19, out1 => #Out_Functional_Test.Electrical_Current_Read_PLC_Functional_Test_19)
   END_RUNG
   RUNG wire#w1
      Contact( #In_Functional_Test.Life_Trigger_PLC_Functional_Test_21 )
      Coil( #Out_Functional_Test.Life_Trigger_PLC_Functional_Test_21 )
   END_RUNG
   RUNG wire#w1
      Contact( #In_Functional_Test.Star_Test_PLC_Functional_Test_21 )
      Coil( #Out_Functional_Test.Star_Test_PLC_Functional_Test_21 )
   END_RUNG
   RUNG wire#w1
      Contact( #In_Functional_Test.Button_PLC_Functional_Test_21 )
      Coil( #Out_Functional_Test.Button_PLC_Functional_Test_21 )
   END_RUNG
   RUNG wire#w1
      Contact( #In_Functional_Test.Electrical_Current_Test_Approved_PLC_Functional_Test_21 )
      Coil( #Out_Functional_Test.Electrical_Current_Test_Approved_PLC_Functional_Test_21 )
   END_RUNG
   RUNG wire#w1
      Contact( #In_Functional_Test.Visual_Test_Approved_PLC_Functional_Test_21 )
      Coil( #Out_Functional_Test.Visual_Test_Approved_PLC_Functional_Test_21 )
   END_RUNG
   RUNG wire#w1
      Move(in := #In_Functional_Test.Electrical_Current_Read_PLC_Functional_Test_21, out1 => #Out_Functional_Test.Electrical_Current_Read_PLC_Functional_Test_21)
   END_RUNG
   RUNG wire#w1
      Contact( #In_Functional_Test.Life_Trigger_PLC_Functional_Test_23 )
      Coil( #Out_Functional_Test.Life_Trigger_PLC_Functional_Test_23 )
   END_RUNG
   RUNG wire#w1
      Contact( #In_Functional_Test.Star_Test_PLC_Functional_Test_23 )
      Coil( #Out_Functional_Test.Star_Test_PLC_Functional_Test_23 )
   END_RUNG
   RUNG wire#w1
      Contact( #In_Functional_Test.Button_PLC_Functional_Test_23 )
      Coil( #Out_Functional_Test.Button_PLC_Functional_Test_23 )
   END_RUNG
   RUNG wire#w1
      Contact( #In_Functional_Test.Electrical_Current_Test_Approved_PLC_Functional_Test_23 )
      Coil( #Out_Functional_Test.Electrical_Current_Test_Approved_PLC_Functional_Test_23 )
   END_RUNG
   RUNG wire#w1
      Contact( #In_Functional_Test.Visual_Test_Approved_PLC_Functional_Test_23 )
      Coil( #Out_Functional_Test.Visual_Test_Approved_PLC_Functional_Test_23 )
   END_RUNG
   RUNG wire#w1
      Move(in := #In_Functional_Test.Electrical_Current_Read_PLC_Functional_Test_23, out1 => #Out_Functional_Test.Electrical_Current_Read_PLC_Functional_Test_23)
   END_RUNG
   RUNG wire#w1
      Contact( #In_Functional_Test.Life_Trigger_PLC_Functional_Test_25 )
      Coil( #Out_Functional_Test.Life_Trigger_PLC_Functional_Test_25 )
   END_RUNG
   RUNG wire#w1
      Contact( #In_Functional_Test.Star_Test_PLC_Functional_Test_25 )
      Coil( #Out_Functional_Test.Star_Test_PLC_Functional_Test_25 )
   END_RUNG
   RUNG wire#w1
      Contact( #In_Functional_Test.Button_PLC_Functional_Test_25 )
      Coil( #Out_Functional_Test.Button_PLC_Functional_Test_25 )
   END_RUNG
   RUNG wire#w1
      Contact( #In_Functional_Test.Electrical_Current_Test_Approved_PLC_Functional_Test_25 )
      Coil( #Out_Functional_Test.Electrical_Current_Test_Approved_PLC_Functional_Test_25 )
   END_RUNG
   RUNG wire#w1
      Contact( #In_Functional_Test.Visual_Test_Approved_PLC_Functional_Test_25 )
      Coil( #Out_Functional_Test.Visual_Test_Approved_PLC_Functional_Test_25 )
   END_RUNG
   RUNG wire#w1
      Move(in := #In_Functional_Test.Electrical_Current_Read_PLC_Functional_Test_25, out1 => #Out_Functional_Test.Electrical_Current_Read_PLC_Functional_Test_25)
   END_RUNG
   RUNG wire#w1
      Contact( #In_Functional_Test.Life_Trigger_PLC_Functional_Test_27 )
      Coil( #Out_Functional_Test.Life_Trigger_PLC_Functional_Test_27 )
   END_RUNG
   RUNG wire#w1
      Contact( #In_Functional_Test.Star_Test_PLC_Functional_Test_27 )
      Coil( #Out_Functional_Test.Star_Test_PLC_Functional_Test_27 )
   END_RUNG
   RUNG wire#w1
      Contact( #In_Functional_Test.Button_PLC_Functional_Test_27 )
      Coil( #Out_Functional_Test.Button_PLC_Functional_Test_27 )
   END_RUNG
   RUNG wire#w1
      Contact( #In_Functional_Test.Electrical_Current_Test_Approved_PLC_Functional_Test_27 )
      Coil( #Out_Functional_Test.Electrical_Current_Test_Approved_PLC_Functional_Test_27 )
   END_RUNG
   RUNG wire#w1
      Contact( #In_Functional_Test.Visual_Test_Approved_PLC_Functional_Test_27 )
      Coil( #Out_Functional_Test.Visual_Test_Approved_PLC_Functional_Test_27 )
   END_RUNG
   RUNG wire#w1
      Move(in := #In_Functional_Test.Electrical_Current_Read_PLC_Functional_Test_27, out1 => #Out_Functional_Test.Electrical_Current_Read_PLC_Functional_Test_27)
   END_RUNG
   RUNG wire#w1
      Contact( #In_Functional_Test.Life_Trigger_PLC_Functional_Test_29 )
      Coil( #Out_Functional_Test.Life_Trigger_PLC_Functional_Test_29 )
   END_RUNG
   RUNG wire#w1
      Contact( #In_Functional_Test.Star_Test_PLC_Functional_Test_29 )
      Coil( #Out_Functional_Test.Star_Test_PLC_Functional_Test_29 )
   END_RUNG
   RUNG wire#w1
      Contact( #In_Functional_Test.Button_PLC_Functional_Test_29 )
      Coil( #Out_Functional_Test.Button_PLC_Functional_Test_29 )
   END_RUNG
   RUNG wire#w1
      Contact( #In_Functional_Test.Electrical_Current_Test_Approved_PLC_Functional_Test_29 )
      Coil( #Out_Functional_Test.Electrical_Current_Test_Approved_PLC_Functional_Test_29 )
   END_RUNG
   RUNG wire#w1
      Contact( #In_Functional_Test.Visual_Test_Approved_PLC_Functional_Test_29 )
      Coil( #Out_Functional_Test.Visual_Test_Approved_PLC_Functional_Test_29 )
   END_RUNG
   RUNG wire#w1
      Move(in := #In_Functional_Test.Electrical_Current_Read_PLC_Functional_Test_29, out1 => #Out_Functional_Test.Electrical_Current_Read_PLC_Functional_Test_29)
   END_RUNG
   // the same network as SCL:
   #_w1 := #Test_Station = 3;
   #Out_Functional_Test.Life_Trigger_PLC_Functional_Test_3 := #_w1 AND #Life_Trigger;
   #Out_Functional_Test.Star_Test_PLC_Functional_Test_3 := #_w1 AND #Star_Test;
   #Out_Functional_Test.Button_PLC_Functional_Test_3 := #_w1 AND #Button_Start_Approve;
   #Out_Functional_Test.Electrical_Current_Test_Approved_PLC_Functional_Test_3 := #_w1 AND #Electrical_Current_Test_Approved;
   #Out_Functional_Test.Visual_Test_Approved_PLC_Functional_Test_3 := #_w1 AND #Visual_Test_Approved;
   #Reset_Functional_Test := #_w1 AND #In_Test_Parameters.Reset_PLC_Functional_Test_3;
   IF #_w1 THEN
       #Out_Functional_Test.Electrical_Current_Read_PLC_Functional_Test_3 := #Electrical_Current_Read;
   END_IF;
   #Out_Functional_Test.Life_Trigger_PLC_Functional_Test_5 := #_w1 AND #In_Functional_Test.Life_Trigger_PLC_Functional_Test_5;
   #Out_Functional_Test.Star_Test_PLC_Functional_Test_5 := #_w1 AND #In_Functional_Test.Star_Test_PLC_Functional_Test_5;
   #Out_Functional_Test.Button_PLC_Functional_Test_5 := #_w1 AND #In_Functional_Test.Button_PLC_Functional_Test_5;
   #Out_Functional_Test.Electrical_Current_Test_Approved_PLC_Functional_Test_5 := #_w1 AND #In_Functional_Test.Electrical_Current_Test_Approved_PLC_Functional_Test_5;
   #Out_Functional_Test.Visual_Test_Approved_PLC_Functional_Test_5 := #_w1 AND #In_Functional_Test.Visual_Test_Approved_PLC_Functional_Test_5;
   IF #_w1 THEN
       #Out_Functional_Test.Electrical_Current_Read_PLC_Functional_Test_5 := #In_Functional_Test.Electrical_Current_Read_PLC_Functional_Test_5;
   END_IF;
   #Out_Functional_Test.Life_Trigger_PLC_Functional_Test_7 := #_w1 AND #In_Functional_Test.Life_Trigger_PLC_Functional_Test_7;
   #Out_Functional_Test.Star_Test_PLC_Functional_Test_7 := #_w1 AND #In_Functional_Test.Star_Test_PLC_Functional_Test_7;
   #Out_Functional_Test.Button_PLC_Functional_Test_7 := #_w1 AND #In_Functional_Test.Button_PLC_Functional_Test_7;
   #Out_Functional_Test.Electrical_Current_Test_Approved_PLC_Functional_Test_7 := #_w1 AND #In_Functional_Test.Electrical_Current_Test_Approved_PLC_Functional_Test_7;
   #Out_Functional_Test.Visual_Test_Approved_PLC_Functional_Test_7 := #_w1 AND #In_Functional_Test.Visual_Test_Approved_PLC_Functional_Test_7;
   IF #_w1 THEN
       #Out_Functional_Test.Electrical_Current_Read_PLC_Functional_Test_7 := #In_Functional_Test.Electrical_Current_Read_PLC_Functional_Test_7;
   END_IF;
   #Out_Functional_Test.Life_Trigger_PLC_Functional_Test_9 := #_w1 AND #In_Functional_Test.Life_Trigger_PLC_Functional_Test_9;
   #Out_Functional_Test.Star_Test_PLC_Functional_Test_9 := #_w1 AND #In_Functional_Test.Star_Test_PLC_Functional_Test_9;
   #Out_Functional_Test.Button_PLC_Functional_Test_9 := #_w1 AND #In_Functional_Test.Button_PLC_Functional_Test_9;
   #Out_Functional_Test.Electrical_Current_Test_Approved_PLC_Functional_Test_9 := #_w1 AND #In_Functional_Test.Electrical_Current_Test_Approved_PLC_Functional_Test_9;
   #Out_Functional_Test.Visual_Test_Approved_PLC_Functional_Test_9 := #_w1 AND #In_Functional_Test.Visual_Test_Approved_PLC_Functional_Test_9;
   IF #_w1 THEN
       #Out_Functional_Test.Electrical_Current_Read_PLC_Functional_Test_9 := #In_Functional_Test.Electrical_Current_Read_PLC_Functional_Test_9;
   END_IF;
   #Out_Functional_Test.Life_Trigger_PLC_Functional_Test_11 := #_w1 AND #In_Functional_Test.Life_Trigger_PLC_Functional_Test_11;
   #Out_Functional_Test.Star_Test_PLC_Functional_Test_11 := #_w1 AND #In_Functional_Test.Star_Test_PLC_Functional_Test_11;
   #Out_Functional_Test.Button_PLC_Functional_Test_11 := #_w1 AND #In_Functional_Test.Button_PLC_Functional_Test_11;
   #Out_Functional_Test.Electrical_Current_Test_Approved_PLC_Functional_Test_11 := #_w1 AND #In_Functional_Test.Electrical_Current_Test_Approved_PLC_Functional_Test_11;
   #Out_Functional_Test.Visual_Test_Approved_PLC_Functional_Test_11 := #_w1 AND #In_Functional_Test.Visual_Test_Approved_PLC_Functional_Test_11;
   IF #_w1 THEN
       #Out_Functional_Test.Electrical_Current_Read_PLC_Functional_Test_11 := #In_Functional_Test.Electrical_Current_Read_PLC_Functional_Test_11;
   END_IF;
   #Out_Functional_Test.Life_Trigger_PLC_Functional_Test_13 := #_w1 AND #In_Functional_Test.Life_Trigger_PLC_Functional_Test_13;
   #Out_Functional_Test.Star_Test_PLC_Functional_Test_13 := #_w1 AND #In_Functional_Test.Star_Test_PLC_Functional_Test_13;
   #Out_Functional_Test.Button_PLC_Functional_Test_13 := #_w1 AND #In_Functional_Test.Button_PLC_Functional_Test_13;
   #Out_Functional_Test.Electrical_Current_Test_Approved_PLC_Functional_Test_13 := #_w1 AND #In_Functional_Test.Electrical_Current_Test_Approved_PLC_Functional_Test_13;
   #Out_Functional_Test.Visual_Test_Approved_PLC_Functional_Test_13 := #_w1 AND #In_Functional_Test.Visual_Test_Approved_PLC_Functional_Test_13;
   IF #_w1 THEN
       #Out_Functional_Test.Electrical_Current_Read_PLC_Functional_Test_13 := #In_Functional_Test.Electrical_Current_Read_PLC_Functional_Test_13;
   END_IF;
   #Out_Functional_Test.Life_Trigger_PLC_Functional_Test_15 := #_w1 AND #In_Functional_Test.Life_Trigger_PLC_Functional_Test_15;
   #Out_Functional_Test.Star_Test_PLC_Functional_Test_15 := #_w1 AND #In_Functional_Test.Star_Test_PLC_Functional_Test_15;
   #Out_Functional_Test.Button_PLC_Functional_Test_15 := #_w1 AND #In_Functional_Test.Button_PLC_Functional_Test_15;
   #Out_Functional_Test.Electrical_Current_Test_Approved_PLC_Functional_Test_15 := #_w1 AND #In_Functional_Test.Electrical_Current_Test_Approved_PLC_Functional_Test_15;
   #Out_Functional_Test.Visual_Test_Approved_PLC_Functional_Test_15 := #_w1 AND #In_Functional_Test.Visual_Test_Approved_PLC_Functional_Test_15;
   IF #_w1 THEN
       #Out_Functional_Test.Electrical_Current_Read_PLC_Functional_Test_15 := #In_Functional_Test.Electrical_Current_Read_PLC_Functional_Test_15;
   END_IF;
   #Out_Functional_Test.Life_Trigger_PLC_Functional_Test_17 := #_w1 AND #In_Functional_Test.Life_Trigger_PLC_Functional_Test_17;
   #Out_Functional_Test.Star_Test_PLC_Functional_Test_17 := #_w1 AND #In_Functional_Test.Star_Test_PLC_Functional_Test_17;
   #Out_Functional_Test.Button_PLC_Functional_Test_17 := #_w1 AND #In_Functional_Test.Button_PLC_Functional_Test_17;
   #Out_Functional_Test.Electrical_Current_Test_Approved_PLC_Functional_Test_17 := #_w1 AND #In_Functional_Test.Electrical_Current_Test_Approved_PLC_Functional_Test_17;
   #Out_Functional_Test.Visual_Test_Approved_PLC_Functional_Test_17 := #_w1 AND #In_Functional_Test.Visual_Test_Approved_PLC_Functional_Test_17;
   IF #_w1 THEN
       #Out_Functional_Test.Electrical_Current_Read_PLC_Functional_Test_17 := #In_Functional_Test.Electrical_Current_Read_PLC_Functional_Test_17;
   END_IF;
   #Out_Functional_Test.Life_Trigger_PLC_Functional_Test_19 := #_w1 AND #In_Functional_Test.Life_Trigger_PLC_Functional_Test_19;
   #Out_Functional_Test.Star_Test_PLC_Functional_Test_19 := #_w1 AND #In_Functional_Test.Star_Test_PLC_Functional_Test_19;
   #Out_Functional_Test.Button_PLC_Functional_Test_19 := #_w1 AND #In_Functional_Test.Button_PLC_Functional_Test_19;
   #Out_Functional_Test.Electrical_Current_Test_Approved_PLC_Functional_Test_19 := #_w1 AND #In_Functional_Test.Electrical_Current_Test_Approved_PLC_Functional_Test_19;
   #Out_Functional_Test.Visual_Test_Approved_PLC_Functional_Test_19 := #_w1 AND #In_Functional_Test.Visual_Test_Approved_PLC_Functional_Test_19;
   IF #_w1 THEN
       #Out_Functional_Test.Electrical_Current_Read_PLC_Functional_Test_19 := #In_Functional_Test.Electrical_Current_Read_PLC_Functional_Test_19;
   END_IF;
   #Out_Functional_Test.Life_Trigger_PLC_Functional_Test_21 := #_w1 AND #In_Functional_Test.Life_Trigger_PLC_Functional_Test_21;
   #Out_Functional_Test.Star_Test_PLC_Functional_Test_21 := #_w1 AND #In_Functional_Test.Star_Test_PLC_Functional_Test_21;
   #Out_Functional_Test.Button_PLC_Functional_Test_21 := #_w1 AND #In_Functional_Test.Button_PLC_Functional_Test_21;
   #Out_Functional_Test.Electrical_Current_Test_Approved_PLC_Functional_Test_21 := #_w1 AND #In_Functional_Test.Electrical_Current_Test_Approved_PLC_Functional_Test_21;
   #Out_Functional_Test.Visual_Test_Approved_PLC_Functional_Test_21 := #_w1 AND #In_Functional_Test.Visual_Test_Approved_PLC_Functional_Test_21;
   IF #_w1 THEN
       #Out_Functional_Test.Electrical_Current_Read_PLC_Functional_Test_21 := #In_Functional_Test.Electrical_Current_Read_PLC_Functional_Test_21;
   END_IF;
   #Out_Functional_Test.Life_Trigger_PLC_Functional_Test_23 := #_w1 AND #In_Functional_Test.Life_Trigger_PLC_Functional_Test_23;
   #Out_Functional_Test.Star_Test_PLC_Functional_Test_23 := #_w1 AND #In_Functional_Test.Star_Test_PLC_Functional_Test_23;
   #Out_Functional_Test.Button_PLC_Functional_Test_23 := #_w1 AND #In_Functional_Test.Button_PLC_Functional_Test_23;
   #Out_Functional_Test.Electrical_Current_Test_Approved_PLC_Functional_Test_23 := #_w1 AND #In_Functional_Test.Electrical_Current_Test_Approved_PLC_Functional_Test_23;
   #Out_Functional_Test.Visual_Test_Approved_PLC_Functional_Test_23 := #_w1 AND #In_Functional_Test.Visual_Test_Approved_PLC_Functional_Test_23;
   IF #_w1 THEN
       #Out_Functional_Test.Electrical_Current_Read_PLC_Functional_Test_23 := #In_Functional_Test.Electrical_Current_Read_PLC_Functional_Test_23;
   END_IF;
   #Out_Functional_Test.Life_Trigger_PLC_Functional_Test_25 := #_w1 AND #In_Functional_Test.Life_Trigger_PLC_Functional_Test_25;
   #Out_Functional_Test.Star_Test_PLC_Functional_Test_25 := #_w1 AND #In_Functional_Test.Star_Test_PLC_Functional_Test_25;
   #Out_Functional_Test.Button_PLC_Functional_Test_25 := #_w1 AND #In_Functional_Test.Button_PLC_Functional_Test_25;
   #Out_Functional_Test.Electrical_Current_Test_Approved_PLC_Functional_Test_25 := #_w1 AND #In_Functional_Test.Electrical_Current_Test_Approved_PLC_Functional_Test_25;
   #Out_Functional_Test.Visual_Test_Approved_PLC_Functional_Test_25 := #_w1 AND #In_Functional_Test.Visual_Test_Approved_PLC_Functional_Test_25;
   IF #_w1 THEN
       #Out_Functional_Test.Electrical_Current_Read_PLC_Functional_Test_25 := #In_Functional_Test.Electrical_Current_Read_PLC_Functional_Test_25;
   END_IF;
   #Out_Functional_Test.Life_Trigger_PLC_Functional_Test_27 := #_w1 AND #In_Functional_Test.Life_Trigger_PLC_Functional_Test_27;
   #Out_Functional_Test.Star_Test_PLC_Functional_Test_27 := #_w1 AND #In_Functional_Test.Star_Test_PLC_Functional_Test_27;
   #Out_Functional_Test.Button_PLC_Functional_Test_27 := #_w1 AND #In_Functional_Test.Button_PLC_Functional_Test_27;
   #Out_Functional_Test.Electrical_Current_Test_Approved_PLC_Functional_Test_27 := #_w1 AND #In_Functional_Test.Electrical_Current_Test_Approved_PLC_Functional_Test_27;
   #Out_Functional_Test.Visual_Test_Approved_PLC_Functional_Test_27 := #_w1 AND #In_Functional_Test.Visual_Test_Approved_PLC_Functional_Test_27;
   IF #_w1 THEN
       #Out_Functional_Test.Electrical_Current_Read_PLC_Functional_Test_27 := #In_Functional_Test.Electrical_Current_Read_PLC_Functional_Test_27;
   END_IF;
   #Out_Functional_Test.Life_Trigger_PLC_Functional_Test_29 := #_w1 AND #In_Functional_Test.Life_Trigger_PLC_Functional_Test_29;
   #Out_Functional_Test.Star_Test_PLC_Functional_Test_29 := #_w1 AND #In_Functional_Test.Star_Test_PLC_Functional_Test_29;
   #Out_Functional_Test.Button_PLC_Functional_Test_29 := #_w1 AND #In_Functional_Test.Button_PLC_Functional_Test_29;
   #Out_Functional_Test.Electrical_Current_Test_Approved_PLC_Functional_Test_29 := #_w1 AND #In_Functional_Test.Electrical_Current_Test_Approved_PLC_Functional_Test_29;
   #Out_Functional_Test.Visual_Test_Approved_PLC_Functional_Test_29 := #_w1 AND #In_Functional_Test.Visual_Test_Approved_PLC_Functional_Test_29;
   IF #_w1 THEN
       #Out_Functional_Test.Electrical_Current_Read_PLC_Functional_Test_29 := #In_Functional_Test.Electrical_Current_Read_PLC_Functional_Test_29;
   END_IF;
END_REGION

